Yaskawa INFORM job: SKRZYNIA_4740_0_STOPNI_2OBR.JBI

/JOB
//NAME SKRZYNIA_4740_0_STOPNI_2OBR
///FOLDERNAME 02-SKRZYNIE_JOBS
//POS
///NPOS 698,698,0,50,0,0
///TOOL 0
///POSTYPE PULSE
///PULSE
C00000=1055,-24125,84372,288,19725,204
C00001=0,-15438,65714,0,-68532,0
C00002=4718,-16587,59952,3396,-65485,-935
C00003=32997,-21499,42555,27623,-61436,21376
C00004=31759,-20688,42932,26837,-60850,21559
C00005=28987,-21156,42712,24818,-60442,22222
C00006=33447,-21964,42352,27886,-61721,21330
C00007=37687,-23357,41794,30651,-63289,20620
C00008=38979,-19018,48057,32961,-64962,20678
C00009=37261,-18075,48526,31902,-64209,20901
C00010=35830,-17198,48994,31015,-63571,21092
C00011=34080,-17614,48768,29780,-63290,21485
C00012=37261,-18075,48526,31902,-64209,20901
C00013=4718,-16587,59952,3396,-65485,-935
C00014=32997,-21499,42555,27623,-61436,21376
C00015=31759,-20688,42932,26837,-60850,21559
C00016=28987,-21156,42712,24818,-60442,22222
C00017=33447,-21964,42352,27886,-61721,21330
C00018=37687,-23357,41794,30651,-63289,20620
C00019=38979,-19018,48057,32961,-64962,20678
C00020=37261,-18075,48526,31902,-64209,20901
C00021=35830,-17198,48994,31015,-63571,21092
C00022=34080,-17614,48768,29780,-63290,21485
C00023=37261,-18075,48526,31902,-64209,20901
C00024=47373,-21912,40596,41149,-66086,26950
C00025=45033,-20851,41104,39798,-65001,27223
C00026=42790,-19693,41704,38494,-63946,27495
C00027=41070,-20182,41442,37324,-63566,27891
C00028=45033,-20851,41104,39798,-65001,27223
C00029=45033,-20851,41104,39798,-65001,27223
C00030=59624,-29540,14278,64846,-60867,16042
C00031=57357,-28542,14780,63940,-59509,16120
C00032=56188,-29140,14476,63237,-58995,16387
C00033=59588,-29370,14363,64862,-60819,16012
C00034=70875,-38414,-12574,117781,-105744,5605
C00035=70875,-38414,-12574,117781,-105744,5605
C00036=58486,-39981,-10562,86359,-50427,5279
C00037=56769,-35832,-2792,84059,-49443,6631
C00038=55152,-35009,-2405,83835,-48426,6454
C00039=53661,-35722,-2740,83085,-47530,6682
C00040=56769,-35832,-2792,84059,-49443,6631
C00041=87562,-48087,-13810,78020,-75252,11220
C00042=10104,-46603,4759,11228,-37390,-5046
C00043=0,-52280,40443,0,6876,0
C00044=1529,-42140,58025,-5964,2417,3265
C00045=0,-38374,23626,-1605,-51738,268
C00046=45044,-23015,37260,35797,-71879,25522
C00047=39973,-29571,18873,35060,-63052,24165
C00048=38620,-28701,19269,34339,-62304,24363
C00049=36409,-29254,19014,32896,-61805,24958
C00050=44451,-29039,21934,37281,-65892,23702
C00051=49472,-39353,6917,53118,-50908,20251
C00052=45058,-39356,3832,51653,-47640,20099
C00053=42883,-38319,4163,50577,-46309,20295
C00054=40255,-38926,3967,48502,-45334,21060
C00055=46774,-39679,3737,52663,-48537,19827
C00056=48708,-40455,3517,53615,-49689,19657
C00057=43798,-39237,3871,50850,-47027,20335
C00058=41951,-38324,4161,49930,-45891,20507
C00059=39836,-38844,3994,48234,-45126,21137
C00060=48489,-40338,3551,53521,-49551,19665
///LIMIT ON
C00061=1148,-56354,34370,-23,3827,-9
C00062=1148,-56354,34370,-23,3827,-9
///LIMIT OFF
C00063=48489,-40338,3551,53521,-49551,19665
C00064=44432,-39026,3936,51363,-47247,20139
C00065=42487,-38069,4248,50403,-46050,20315
C00066=39061,-38795,4009,47695,-44769,21310
C00067=44432,-39026,3936,51363,-47247,20139
C00068=43521,-36748,12770,50182,-45701,23408
C00069=41846,-35383,13175,49516,-44517,23399
C00070=39971,-34448,13485,48491,-43408,23582
C00071=37453,-34980,13306,46330,-42542,24334
C00072=41846,-35383,13175,49516,-44517,23399
C00073=78369,-41260,16071,67181,-65880,21417
C00074=137,-45861,52341,97,-67596,-14
C00075=-31499,-58302,-23356,15027,12889,-13082
C00076=-52768,-43016,-26078,18373,38595,-18774
C00077=-89470,-32103,-32973,29905,69139,-31512
C00078=-68838,-26884,-24872,16972,64732,-23076
C00079=-53036,-11528,-12218,12363,64665,-17409
C00080=-51536,-9474,-10276,11905,64649,-16876
C00081=-51739,-9114,-7787,12104,63269,-17104
C00082=-53036,-11528,-12218,12363,64665,-17409
C00083=-17541,-26226,-24397,927,59032,-5038
C00084=-17541,-26226,-24397,927,59032,-5038
C00085=-16950,-23991,-22741,715,59568,-4818
C00086=-17036,-23563,-20101,755,58071,-4857
C00087=-17541,-26226,-24397,927,59032,-5038
C00088=34102,-23192,-21614,-15638,64271,13209
C00089=33423,-21885,-20599,-15423,64418,12942
C00090=32426,-19856,-18975,-15106,64629,12551
C00091=32578,-19611,-17013,-15290,63535,12762
C00092=33423,-21885,-20599,-15423,64418,12942
C00093=59339,-6070,-6417,-20979,72191,20891
C00094=59339,-6070,-6417,-20979,72191,20891
C00095=57897,-4256,-4562,-20702,71913,20431
C00096=58108,-3992,-2506,-20878,70835,20713
C00097=59339,-6070,-6417,-20979,72191,20891
C00098=42744,-35904,-30225,-18322,62562,16651
C00099=-53036,-11528,-12218,12363,64665,-17409
C00100=-77982,-26538,-29134,27151,66629,-27745
C00101=-70983,-8594,-1966,26503,59809,-49670
C00102=-80152,19776,40785,37351,72704,-50428
C00103=-79984,20154,42529,37516,71911,-50638
C00104=-79233,18397,40079,37458,71885,-50340
C00105=-79984,20154,42529,37516,71911,-50638
C00106=-73519,23289,38838,28890,77081,-45618
C00107=-73519,24511,42682,29072,75582,-46027
C00108=-73519,23289,38838,28890,77081,-45618
C00109=-88897,15706,42282,50101,71325,-56974
C00110=-88897,15706,42282,50101,71325,-56974
C00111=-87612,12343,37838,50071,70996,-56519
C00112=-85283,14202,40272,50301,69633,-56165
C00113=-87338,12550,38107,50098,70839,-56476
C00114=-84952,-1789,13569,34660,47724,-58955
C00115=-67641,-1674,11109,10330,44856,-44725
C00116=-66443,961,13975,9688,44721,-44210
C00117=-67641,-1674,11109,10330,44856,-44725
C00118=-67641,-376,15347,10694,42950,-44967
C00119=-67641,-1674,11109,10330,44856,-44725
C00120=-79040,417,20398,15965,28992,-57786
C00121=-76655,5212,30978,15501,25024,-57306
C00122=-76655,6949,35816,16758,23084,-57955
C00123=-76655,5212,30978,15501,25024,-57306
C00124=-74761,6919,33010,13466,24593,-56049
C00125=-80460,-2874,12270,15804,32253,-57809
C00126=-61258,-29124,-13156,26560,43617,-22150
C00127=-30420,-40507,-29240,27153,53235,15188
C00128=-18589,-38725,-21450,23338,47896,18931
C00129=-17722,-35233,-16455,23322,46926,19051
C00130=-17722,-33749,-12435,23948,45421,18620
C00131=-17722,-33892,-12819,23887,45564,18661
C00132=-16677,-31133,-11209,23138,46167,19311
C00133=-17819,-35820,-17540,23246,47228,19090
C00134=-74104,-11494,-6266,31916,75042,4269
C00135=-71226,-7329,2631,32115,71468,4273
C00136=-71226,-6504,5446,32343,70365,3922
C00137=-71226,-6611,5086,32313,70505,3967
C00138=-68386,-4058,7675,32040,69573,4789
C00139=-73314,-9412,-353,32206,72648,3829
C00140=51751,-31069,-22965,-10739,49070,48663
C00141=49028,-23852,-11575,-9841,46366,47823
C00142=49028,-23004,-8935,-10039,45204,47956
C00143=49028,-23118,-9286,-10013,45357,47939
C00144=47000,-20813,-7527,-8928,45644,47024
C00145=50476,-26208,-15307,-10408,47325,48332
C00146=90602,-5375,6902,-38786,69848,59444
C00147=83174,19950,50269,-44999,67580,58220
C00148=82362,17902,47383,-44926,67511,57879
C00149=83515,19072,48341,-44798,68200,58056
C00150=78091,19382,40247,-36371,72286,52960
C00151=78091,20664,44011,-36670,70997,53443
C00152=78091,19382,40247,-36371,72286,52960
C00153=88699,7296,38566,-55615,63182,60372
C00154=86803,3068,32674,-55410,62638,59657
C00155=84852,4315,34115,-55564,61561,59330
C00156=86803,3068,32674,-55410,62638,59657
C00157=92770,-2803,21719,-53893,67577,59421
C00158=73393,-10627,10934,-27897,30744,62458
C00159=70789,-6606,18800,-27824,27830,62140
C00160=69654,-4593,20814,-26755,27596,61444
C00161=70789,-6606,18800,-27824,27830,62140
C00162=70789,-5070,23059,-29482,26284,63017
C00163=70789,-6606,18800,-27824,27830,62140
C00164=83486,-8736,6503,-27040,35338,66550
C00165=77831,-2041,26192,-25270,18452,68895
C00166=77967,1961,32070,-26860,17569,69698
C00167=77967,5243,40752,-32914,14549,72656
C00168=77967,1961,32070,-26860,17569,69698
C00169=74560,4730,35257,-21622,16551,66717
C00170=77967,1961,32070,-26860,17569,69698
C00171=81109,-22356,2664,-22493,33121,60116
C00172=86168,-49730,-13668,-23926,46819,49343
C00173=44183,-52048,-7537,-24795,46064,51426
C00174=0,-52280,40443,0,6876,0
C00175=0,-52280,40443,0,6876,0
C00176=33629,-57276,-6399,46271,-24969,-2804
C00177=75493,-63502,-64712,103874,-64610,-6298
C00178=48303,-58663,-62781,109560,-46378,-10551
C00179=44029,-59891,-64997,113806,-43206,-9136
C00180=55379,-67378,-68041,108237,-48773,-4935
C00181=62671,-64213,-64640,104431,-56093,-7372
C00182=28458,-50318,6850,47420,-25887,-3347
C00183=0,-52280,40443,0,6876,0
C00184=1055,-24125,84372,288,19725,204
C00185=0,-15438,65714,0,-68532,0
C00186=0,-15438,65714,966,-70097,42926
C00187=69988,-9219,57065,61610,-82752,27767
C00188=63113,-6157,59685,58080,-79692,28271
C00189=46529,-7301,64143,40614,-74233,29269
C00190=49501,-5951,66049,43527,-75687,29381
C00191=53417,-8187,64183,45775,-77170,28968
C00192=63113,-6157,59685,58080,-79692,28271
C00193=69988,-9219,57065,61610,-82752,27767
C00194=0,-15438,65714,966,-70097,42926
C00195=0,-15438,65714,0,-68532,0
C00196=1055,-24125,84372,288,19725,204
C00197=1055,-24125,84372,288,19725,204
C00198=0,-41971,13909,0,6774,1
C00199=-55064,-17017,13106,20113,45767,-35735
C00200=-85641,-3161,12660,31281,67420,-55579
C00201=-77611,9747,38455,32702,57795,-55547
C00202=-77611,9747,38455,32702,57795,-55547
C00203=-80481,23547,61641,37204,60115,-56891
C00204=-80479,11681,28780,33754,71138,-52780
C00205=-73572,15026,34389,33675,67405,-51294
C00206=-73572,20195,49236,35290,62248,-53161
C00207=-82806,26311,53816,38180,73291,-53604
C00208=-71695,3747,16001,30713,64750,-51022
C00209=-70421,5575,20105,30867,63066,-51036
C00210=-35543,-20105,-5144,22821,50284,-40173
C00211=-37830,-23193,-8618,23571,50957,-40982
C00212=11136,-28839,-12562,1025,41780,-20887
C00213=20486,-27077,-7346,-12554,38415,-10736
C00214=59545,-9921,5571,-27063,51925,3267
C00215=55110,-17412,-5825,-19778,50988,-2825
C00216=79390,11759,28162,-35512,71262,52960
C00217=74811,13878,33986,-35807,67493,52464
C00218=74942,18762,48004,-37392,62815,54352
C00219=76815,18630,46530,-37158,64288,54543
C00220=79390,11759,28162,-35512,71262,52960
C00221=10831,-54278,-29128,-6468,39852,-5090
C00222=-67200,-10549,24402,-3189,24913,-39001
C00223=-75122,-2194,12822,3152,39225,-43427
C00224=-77516,10189,32861,8493,33365,-45533
C00225=-75154,17575,49272,7885,27457,-44928
C00226=-68113,9932,38901,1157,28472,-40453
C00227=-67114,5383,31515,9208,32648,-43213
C00228=-66450,3998,29285,10896,33890,-43630
C00229=-66374,3101,28136,14657,35566,-44954
C00230=-66576,452,24763,27028,43375,-49112
C00231=-69928,4230,30673,35488,50431,-52676
C00232=-77050,-3138,8526,33226,61087,-51698
C00233=-67200,-10549,24402,-3189,24913,-39001
C00234=0,-52280,40443,83103,28146,-16510
C00235=99993,-20782,22705,-13349,24734,56519
C00236=67200,-10549,24402,3189,24913,39001
C00237=75122,-2194,12822,-3152,39225,43427
C00238=74323,5203,27259,-5972,33194,43789
C00239=74015,16414,48063,-6821,27325,44224
C00240=56519,1138,28747,9235,29393,33453
C00241=55467,619,28251,10155,29461,32830
C00242=56374,-724,25854,4078,30541,35419
C00243=56480,-7201,15910,-17697,38451,43334
C00244=68252,956,25699,-34035,49810,51639
C00245=77050,-3138,8526,-33226,61087,51698
C00246=67200,-10549,24402,3189,24913,39001
C00247=0,-52280,40443,-83103,28146,16510
C00248=-99993,-20782,22705,13349,24734,-56519
C00249=-91125,453,39555,30378,52425,-51131
C00250=-81425,-5449,14825,37552,56592,-47667
C00251=-81425,-10835,-2515,34915,62871,-45127
C00252=-79239,4305,16082,37593,68846,-50182
C00253=-81302,5892,27588,46359,62943,-54679
C00254=-82227,19402,59913,51524,57300,-60581
C00255=-84844,8890,27031,38640,69740,-53449
C00256=-90096,4679,14083,37467,76581,-51973
C00257=-87885,29238,52923,40761,81198,69685
C00258=-84355,23847,39024,40698,83720,72224
C00259=-81960,27335,46957,41070,80536,71891
C00260=-82643,24718,50492,48951,72637,70260
C00261=-90480,18737,31939,47254,81986,71631
C00262=-94217,10634,17426,46901,86469,-59967
C00263=-81425,-10835,-2515,34915,62871,-45127
C00264=-81425,-5449,14825,37552,56592,-47667
C00265=-94290,-610,44819,32366,49686,-53459
C00266=0,-55136,17047,60468,32096,-4233
C00267=99993,-20782,22705,-13349,24734,56519
C00268=91125,453,39555,-30378,52425,51131
C00269=81425,-5449,14825,-37552,56592,47667
C00270=81425,-10835,-2515,-34915,62871,45127
C00271=79239,4305,16082,-37593,68846,50182
C00272=83239,4964,30263,-50637,62037,57149
C00273=83991,16425,61235,-57769,55250,63273
C00274=93928,7973,40920,-53095,64494,61640
C00275=75109,22299,39152,-26915,78743,47998
C00276=79256,17348,34699,-33448,76412,88212
C00277=79932,23608,50901,-39863,71219,88955
C00278=76220,30771,63034,-41386,67395,88927
C00279=86322,16060,37848,-39554,76452,89287
C00280=87424,-1569,9538,-38190,72401,52253
C00281=81425,-10835,-2515,-34915,62871,45127
C00282=92850,-11266,9233,-39092,60986,50964
C00283=28366,-40369,19479,-5635,23506,17663
C00284=-80334,-19501,31260,21216,42469,-40219
C00285=-80621,-32280,-9061,25825,59412,-41877
C00286=-80621,-37319,-22868,24573,64555,-40576
C00287=-75108,-2453,16462,35304,60348,-42510
C00288=-72231,7240,33473,36511,55681,-43130
C00289=-35770,-19109,7486,28512,40799,-31761
C00290=-39606,-22901,-1163,28356,44724,-32188
C00291=15344,-29112,-5358,-2858,33820,-6852
C00292=13390,-24012,2637,-1527,32105,-7853
C00293=57983,-8601,15571,-27088,42703,12849
C00294=60973,-17187,4937,-27817,44388,13718
C00295=60973,-17187,4937,-27817,44388,13718
C00296=-13287,-42463,-12044,19170,31021,-23010
C00297=-17374,-21287,20534,22794,29118,-26096
C00298=13276,-20759,18622,-1911,29377,-7028
C00299=39924,-14247,19329,-14795,35999,4396
C00300=41528,-14133,18797,-15449,36702,5040
C00301=57001,-5890,26499,-21893,40771,11494
C00302=64054,-19541,3059,-29141,44956,15011
C00303=51466,-33957,-1499,-46586,51805,23434
C00304=17032,-20770,22044,-28854,30468,11088
C00305=-9868,-18638,14971,-8492,38486,-5199
C00306=-40562,-13194,19800,9508,35447,-20184
C00307=-41848,-12620,20103,10165,35810,-20773
C00308=-57278,-4046,28217,17578,39066,-27653
C00309=-71680,-19835,10874,33863,39440,-36917
C00310=-20806,-37586,-12792,9951,42782,-18031
C00311=29087,-45372,27330,-13325,19529,9021
C00312=0,-52280,40443,0,6876,0
C00313=0,-52280,40443,0,6876,0
C00314=0,-52280,40443,0,6876,0
C00315=0,-52280,40443,0,-40718,0
C00316=32359,-35955,27464,28918,-49457,29587
C00317=33244,-30989,28192,31082,-46894,28340
C00318=17779,-48456,-23364,103225,-11582,-7642
C00319=21302,-27483,32723,20378,-44693,31826
C00320=26032,-39616,1147,25257,-48263,28480
C00321=26032,-42284,-4858,26096,-46359,27892
C00322=29904,-46498,-2819,27004,-47536,28031
C00323=45803,-31685,22885,64496,-39050,18987
C00324=0,-52277,40442,0,6872,2
///LIMIT ON
C00325=0,-38538,66749,0,-898,0
///LIMIT OFF
C00326=0,-52280,40443,0,-79033,35417
C00327=63837,-43435,-10267,65210,-58810,8342
C00328=51738,-38814,-970,57660,-53573,11589
C00329=47613,-40374,-5302,59887,-48365,10192
C00330=46201,-27302,20507,44767,-62342,18270
C00331=53914,-29436,22058,48262,-67266,17843
C00332=63113,-6157,59685,58080,-79692,28271
C00333=53636,-7999,65947,44587,-77595,28821
C00334=47087,-5642,67901,40734,-75391,29611
C00335=49534,-5270,67671,43393,-76105,29552
C00336=58547,-7653,65645,48613,-79176,28479
C00337=0,-52280,40443,0,-79033,35417
C00338=0,-38922,70509,0,-71891,28081
C00339=0,-38922,70509,0,-71891,28081
C00340=36958,-10079,72709,30464,-66560,20948
C00341=30207,-8205,71936,26080,-63666,21556
C00342=5819,-37145,831,436,-53029,28466
C00343=13946,-45192,10090,9828,-39459,25958
///LIMIT ON
C00344=404,-42897,57020,-1574,2523,869
///LIMIT OFF
C00345=0,-52280,40443,0,6876,0
C00346=-99253,-13690,44082,59847,13407,-31313
C00347=-87814,-12734,20141,45739,-14352,-64418
C00348=-86669,-6582,30812,41148,-16781,-62025
C00349=-85055,-5827,31548,44003,-17420,-63187
C00350=-85971,-6262,31124,42409,-17052,-62539
C00351=-86650,-5303,32069,41395,-16716,-62141
C00352=-94954,-14494,-1860,-7818,15857,-59130
C00353=-94509,1544,30797,-849,15127,-60471
C00354=-94509,4151,37772,-1041,12286,-60378
C00355=-88011,-10036,27574,37950,-16527,-60658
C00356=-86125,-12470,22545,29004,-25567,-58412
C00357=-85732,-21202,11427,30682,-24763,-59235
C00358=-84150,-10929,23786,31981,-25941,-59678
C00359=-83036,-10419,24246,33504,-26268,-60308
C00360=-84150,-10929,23786,31981,-25941,-59678
C00361=-85291,-9507,25078,30650,-25411,-59154
C00362=-84150,-10929,23786,31981,-25941,-59678
C00363=-85786,-16909,14677,31743,-23900,-59790
C00364=-84150,-10498,24888,31517,-26306,-59436
C00365=-83174,-10052,25293,32841,-26587,-59984
C00366=-84150,-10498,24888,31517,-26306,-59436
C00367=-85258,-9112,26156,30226,-25800,-58928
C00368=-84150,-10498,24888,31517,-26306,-59436
C00369=-87841,-18519,13420,28367,-23534,-58339
C00370=-84150,-10465,24972,31484,-26336,-59417
C00371=-83241,-10052,25348,32714,-26598,-59924
C00372=-84150,-10465,24972,31484,-26336,-59417
C00373=-85145,-9228,26102,30329,-25881,-58963
C00374=-84150,-10465,24972,31484,-26336,-59417
C00375=-86371,-18277,13606,30568,-23951,-59265
C00376=-84345,-11688,21985,32461,-25312,-59957
C00377=-83211,-11173,22442,34044,-25650,-60618
C00378=-84345,-11688,21985,32461,-25312,-59957
C00379=-85283,-10526,23025,31366,-24861,-59525
C00380=-84345,-11688,21985,32461,-25312,-59957
C00381=-86191,-19647,12567,30467,-24278,-59187
C00382=-84345,-10877,24073,31552,-26006,-59481
C00383=-83051,-10286,24607,33321,-26381,-60213
C00384=-84345,-10877,24073,31552,-26006,-59481
C00385=-85179,-9842,25009,30582,-25619,-59100
C00386=-84345,-10877,24073,31552,-26006,-59481
C00387=-85438,-18022,14839,31140,-24818,-59429
C00388=-84247,-11820,22550,32049,-25753,-59727
C00389=-84104,-10976,23642,32111,-25899,-59738
C00390=-82990,-10465,24105,33639,-26227,-60372
C00391=-84104,-10976,23642,32111,-25899,-59738
C00392=-84898,-9998,24525,31196,-25529,-59378
C00393=-84104,-10976,23642,32111,-25899,-59738
C00394=-86610,-16845,14732,30573,-23614,-59301
C00395=-84104,-10864,23927,31990,-25993,-59674
C00396=-82824,-10273,24459,33737,-26370,-60397
C00397=-84104,-10864,23927,31990,-25993,-59674
C00398=-84789,-10021,24690,31200,-25673,-59363
C00399=-84104,-10864,23927,31990,-25993,-59674
C00400=-83806,-19585,12613,33764,-25080,-60559
C00401=-83924,-10205,25475,31619,-26533,-59453
C00402=-82780,-9675,25960,33156,-26866,-60087
C00403=-83924,-10205,25475,31619,-26533,-59453
C00404=-84478,-9530,26093,30986,-26280,-59206
C00405=-83924,-10205,25475,31619,-26533,-59453
C00406=-87149,-17993,13826,29513,-23647,-58830
C00407=-84920,-13182,20975,31162,-25481,-59361
C00408=-83711,-10572,24852,32056,-26475,-59649
C00409=-82779,-10142,25241,33309,-26748,-60166
C00410=-83711,-10572,24852,32056,-26475,-59649
C00411=-84370,-9774,25579,31305,-26170,-59356
C00412=-83711,-10572,24852,32056,-26475,-59649
C00413=-83642,-3679,42021,23358,-36761,-56118
C00414=-85886,-5975,41264,18964,-40261,-54782
C00415=-83919,-11632,22322,32811,-25616,-60079
C00416=-82884,-11162,22742,34234,-25925,-60671
C00417=-83919,-11632,22322,32811,-25616,-60079
C00418=-84723,-10654,23196,31887,-25230,-59715
C00419=-83919,-11632,22322,32811,-25616,-60079
C00420=-87348,-16035,7353,17528,-35245,-56477
C00421=-86244,-15062,8172,18754,-35315,-57058
C00422=-86244,-16649,3638,19674,-33501,-57585
C00423=-85308,-16228,3988,20718,-33648,-58082
C00424=-86244,-16649,3638,19674,-33501,-57585
C00425=-86740,-15973,4201,19194,-33277,-57362
C00426=-86244,-16649,3638,19674,-33501,-57585
C00427=-73780,-8639,20128,34258,-51705,-52097
C00428=-90711,-17528,-28778,11328,-28245,-57111
C00429=-92565,-19610,-33223,7138,-24591,-57051
C00430=-91512,-19116,-32812,8551,-24603,-57834
C00431=-92565,-19610,-33223,7138,-24591,-57051
C00432=-93003,-18716,-32476,6600,-24397,-56752
C00433=-92565,-19610,-33223,7138,-24591,-57051
C00434=-92565,-19610,-33223,7138,-24591,-57051
C00435=-95836,-54375,-51122,6031,-17685,-48210
C00436=-95836,-54375,-51122,6031,-17685,-48210
C00437=-71303,-59965,-23787,8701,20788,-26710
C00438=-43821,-47238,-2775,-3022,56549,-3681
C00439=-20126,-26882,59542,2406,16879,-9162
C00440=-20126,-26882,59542,2406,16879,-9162
C00441=98601,-10520,92678,4674,-40855,-9615
C00442=95537,-19831,-2695,-2933,-44471,35837
C00443=92548,-20391,-28429,-6186,-30623,55200
C00444=91429,-17018,-28974,-8057,-27827,56250
C00445=91429,-17018,-28974,-8057,-27827,56250
C00446=90371,-16495,-28521,-9286,-27856,56953
C00447=91429,-17018,-28974,-8057,-27827,56250
C00448=92033,-15799,-27911,-7415,-27588,55880
C00449=91429,-17018,-28974,-8057,-27827,56250
C00450=92548,-20391,-28429,-6186,-30623,55200
C00451=91156,-15018,-4648,-8036,-38181,54813
C00452=90585,-14766,-4428,-8565,-38201,55100
C00453=88830,-13959,-3717,-10186,-38284,55977
C00454=89897,-14456,-4157,-9202,-38230,55445
C00455=90761,-12944,-2809,-8452,-37927,55043
C00456=89897,-14456,-4157,-9202,-38230,55445
C00457=89670,-8466,73559,-9449,-60959,55261
C00458=89910,-11217,67535,-9455,-58896,55399
C00459=85786,-16735,14816,-31782,-23869,59812
C00460=83514,-12996,17929,-35760,-24132,61552
C00461=82251,-12406,18443,-37550,-24551,62308
C00462=83514,-12996,17929,-35760,-24132,61552
C00463=84258,-12095,18717,-34917,-23742,61217
C00464=83514,-12996,17929,-35760,-24132,61552
C00465=87149,-17993,13826,-29513,-23647,58830
C00466=83118,-12818,18089,-36330,-24263,61791
C00467=81915,-12248,18589,-38020,-24666,62504
C00468=83118,-12818,18089,-36330,-24263,61791
C00469=83897,-11882,18912,-35460,-23856,61445
C00470=83118,-12818,18089,-36330,-24263,61791
C00471=83806,-19585,12613,-33764,-25080,60559
C00472=82998,-13006,17925,-36445,-24332,61826
C00473=81675,-12378,18472,-38297,-24777,62607
C00474=82998,-13006,17925,-36445,-24332,61826
C00475=83876,-11958,18841,-35466,-23874,61442
C00476=82998,-13006,17925,-36445,-24332,61826
C00477=86610,-16845,14732,-30573,-23614,59301
C00478=82493,-13239,17725,-37070,-24559,62089
C00479=81406,-12724,18174,-38578,-24928,62723
C00480=82493,-13239,17725,-37070,-24559,62089
C00481=83436,-12134,18690,-36041,-24064,61684
C00482=82493,-13239,17725,-37070,-24559,62089
C00483=84814,-16043,15376,-33312,-24093,60464
C00484=82555,-13613,17404,-36910,-24580,62015
C00485=81384,-13062,17878,-38534,-24974,62698
C00486=82555,-13613,17404,-36910,-24580,62015
C00487=83566,-12434,18427,-35805,-24047,61580
C00488=82555,-13613,17404,-36910,-24580,62015
C00489=86191,-19647,12567,-30467,-24278,59187
C00490=82500,-13648,17375,-36975,-24607,62039
C00491=81467,-13161,17792,-38413,-24955,62645
C00492=82500,-13648,17375,-36975,-24607,62039
C00493=83481,-12505,18364,-35905,-24087,61617
C00494=82500,-13648,17375,-36975,-24607,62039
C00495=86371,-18277,13606,-30568,-23951,59265
C00496=82904,-13790,17251,-36416,-24470,61808
C00497=81715,-13237,17726,-38081,-24865,62509
C00498=82904,-13790,17251,-36416,-24470,61808
C00499=83686,-12878,18037,-35556,-24055,61469
C00500=82904,-13790,17251,-36416,-24470,61808
C00501=87841,-18519,13420,-28367,-23534,58339
C00502=82748,-13879,17174,-36603,-24542,61883
C00503=81692,-13388,17594,-38077,-24893,62505
C00504=82748,-13879,17174,-36603,-24542,61883
C00505=83607,-12881,18032,-35663,-24082,61515
C00506=82748,-13879,17174,-36603,-24542,61883
C00507=85786,-16909,14677,-31743,-23900,59790
C00508=82520,-14198,16902,-36833,-24674,61972
C00509=81460,-13708,17319,-38301,-25026,62591
C00510=82520,-14198,16902,-36833,-24674,61972
C00511=83571,-12989,17938,-35691,-24113,61524
C00512=82520,-14198,16902,-36833,-24674,61972
C00513=85732,-21202,11427,-30682,-24763,59235
C00514=82398,-14365,16763,-36952,-24745,62014
C00515=81172,-13798,17245,-38643,-25153,62725
C00516=82398,-14365,16763,-36952,-24745,62014
C00517=83600,-12984,17944,-35650,-24102,61504
C00518=82398,-14365,16763,-36952,-24745,62014
C00519=86140,-12802,12665,-93523,-10743,85795
C00520=86140,-12802,12665,-93523,-10743,85795
C00521=85030,-12289,13120,-93723,-11463,85776
C00522=86140,-12802,12665,-93523,-10743,85795
C00523=86958,-11660,13681,-94506,-10238,86349
C00524=85239,-16743,-4327,42764,21357,45785
C00525=86674,107,23869,25042,24033,51593
C00526=86674,2327,30134,27824,21680,50173
C00527=87715,-15254,10554,-91589,-9692,85040
C00528=85045,-36869,-4353,-28502,-22832,52282
C00529=0,-24029,84339,0,19981,0
C00530=0,-24029,84339,0,19981,0
C00531=3172,-24246,80980,3465,15913,689
C00532=-86563,-26985,13879,10257,-21548,-45530
C00533=-86191,-19647,12567,30467,-24278,-59187
C00534=-83221,-13587,17636,37793,-25116,-62228
C00535=-91978,-13833,14560,12391,-18633,-51524
C00536=-94992,-13830,14285,1276,-18012,-46664
C00537=-84074,-17488,11256,38660,-23649,-62784
C00538=-73679,-33270,1000,44272,-31600,-64253
///LIMIT ON
C00539=-86926,-60758,23267,6576,1160,-9545
///LIMIT OFF
C00540=0,-52280,40443,0,6876,0
///LIMIT ON
C00541=82475,-58079,26734,835,4084,4444
///LIMIT OFF
C00542=97932,-26840,7691,8784,-23444,42538
C00543=87166,-16607,16322,-25365,-24201,56345
C00544=84699,-11354,21752,-29145,-24735,57949
C00545=84804,-11023,22730,-28561,-25071,57659
C00546=85100,-26994,10417,-24982,-28140,55821
C00547=0,-52280,40443,0,6876,0
C00548=0,-52280,40443,0,6876,0
///LIMIT ON
C00549=-90140,-60305,18108,-2708,1721,-7625
///LIMIT OFF
C00550=-95594,-27428,6866,-4663,-19832,-42154
C00551=-98688,-13767,16447,-18366,-10080,-35766
C00552=-98967,-3050,34440,-28957,-8622,-29685
C00553=-100063,5316,51567,-32262,-10006,-27560
C00554=-94586,18541,64268,-6451,10518,-43578
C00555=-95535,2380,25473,239,27557,-47214
C00556=-91259,3120,34463,-5130,22041,-43946
C00557=-95333,12702,45733,36,21375,-47085
C00558=-99268,-13088,27343,-18620,-14105,-35021
///LIMIT ON
C00559=-90140,-60305,18108,-2708,1721,-7625
///LIMIT OFF
C00560=0,-52280,40443,0,6876,0
///LIMIT ON
C00561=84259,-57935,27522,-3761,3673,6310
///LIMIT OFF
C00562=86507,-39672,4297,-27618,-16640,46340
C00563=73669,-37119,-20783,-92053,-19719,85232
C00564=86539,-20830,1725,-71850,-11773,76853
C00565=90325,-18913,6238,-62161,-7452,70888
///LIMIT ON
C00566=97679,-11879,12650,-55334,4229,66281
///LIMIT OFF
C00567=98389,-8856,11720,-15676,14634,48538
C00568=96255,-748,20886,-3277,24061,38276
C00569=95132,-6008,10010,1655,28777,36730
C00570=94050,-4188,7205,-2481,41508,36662
C00571=98126,4908,16834,-5042,41918,38535
C00572=100487,-9453,-1206,-10413,41328,41147
C00573=96250,-19428,-8283,-4838,27297,37910
C00574=86507,-39672,4297,-27618,-16640,46340
///LIMIT ON
C00575=84259,-57935,27522,-3761,3673,6310
///LIMIT OFF
C00576=0,-52280,40443,0,6876,0
C00577=0,-27933,77061,0,20812,0
C00578=0,-27933,77061,0,20812,0
C00579=0,-52280,40443,0,6876,0
///LIMIT ON
C00580=-91970,-60791,14435,-3343,512,-9412
///LIMIT OFF
C00581=-98647,-24138,10005,-11519,-21203,-39749
C00582=-99883,-13980,22886,-11640,-25090,-40341
C00583=-99702,-9154,61728,-1148,-61809,-40243
C00584=-84328,-13042,29707,23458,-33731,-54641
C00585=-83101,-4179,39208,25894,-34785,-55667
C00586=-82881,-4330,38692,26392,-34479,-55866
C00587=-76259,-18287,26646,31659,-38322,-57579
C00588=-89741,-28009,12101,4461,-28076,-46404
///LIMIT ON
C00589=-91970,-60791,14435,-3343,512,-9412
///LIMIT OFF
C00590=0,-52280,40443,0,6876,0
///LIMIT ON
C00591=91083,-60784,14823,-9043,-825,15173
///LIMIT OFF
C00592=83869,-19403,12921,-33769,-24740,60260
C00593=83869,-19403,12921,-33769,-24740,60260
C00594=83932,-19538,53415,-33663,-71112,60249
C00595=83932,-19538,53415,-33663,-71112,60249
C00596=82480,-12247,21118,-35440,-26416,60009
C00597=82194,-11433,19802,-37650,-25323,61125
C00598=81904,-9374,24711,-35791,-26879,60109
C00599=79790,-20261,14917,-36681,-28829,60258
C00600=76554,-29711,-1870,-46042,-25952,65654
///LIMIT ON
C00601=91083,-60784,14823,-9043,-825,15173
///LIMIT OFF
C00602=0,-52280,40443,0,6876,0
///LIMIT ON
C00603=-91526,-60598,16699,7584,176,-13289
///LIMIT OFF
C00604=-81382,-25890,9219,35455,-25500,-59095
C00605=-86453,-20958,12525,30076,-22568,-57089
C00606=-86589,-16097,16237,31250,-21582,-57704
C00607=-98933,-11298,20505,-13970,-18736,-37953
C00608=-98281,-10965,21163,-11559,-18548,-39330
C00609=-85424,-18472,14402,34409,-22969,-58895
C00610=-74746,-27148,8488,44263,-29128,-62418
C00611=-81326,-27507,8265,35533,-26282,-59001
///LIMIT ON
C00612=-91415,-60262,16631,7870,-73,-13734
///LIMIT OFF
C00613=24,-24029,84339,7,19981,5
C00614=100404,-52373,45687,-1822,14816,-5144
C00615=75939,-26469,7919,-40869,-29645,63133
C00616=81882,-22565,10470,-35355,-26404,61107
C00617=82801,-12246,21732,-34208,-26055,60642
C00618=91824,-10567,23615,-8659,-22197,49820
C00619=96485,-9539,26282,5686,-23135,43736
C00620=77262,-23244,14300,-38922,-31295,61912
C00621=96357,-33562,33410,58602,-23427,10353
C00622=568,-24029,84339,168,19981,112
///LIMIT ON
C00623=-91970,-60791,14435,-3343,512,-9412
///LIMIT OFF
C00624=-98991,-22833,11519,-12824,-17638,-36336
C00625=-86376,-13627,18436,38326,-18406,-58533
C00626=-85581,-10814,20279,41280,-18093,-59893
C00627=-85561,-10517,20811,41029,-18209,-59765
C00628=-86274,-24518,9978,34497,-20333,-56613
C00629=-91684,-53777,2301,20525,-9313,-33684
C00630=-67305,-55044,34987,1504,5690,-2468
C00631=0,-52280,40443,0,6876,0
///LIMIT ON
C00632=77036,-56616,31288,-2531,4707,4197
///LIMIT OFF
C00633=84359,-28321,8817,-32860,-20485,54199
C00634=81156,-16932,14874,-39538,-26422,62851
C00635=93321,-15690,11640,-5466,-17578,48664
C00636=91404,-14588,14576,-11730,-19131,51290
C00637=77970,-27630,4721,-41834,-28549,63607
C00638=81111,-35571,7141,-33980,-21909,52006
///LIMIT ON
C00639=82490,-55811,26416,-6832,1088,10458
///LIMIT OFF
C00640=0,-52280,40443,0,6876,0
C00641=0,-28135,76691,0,20839,0
C00642=0,-28135,76691,0,20839,0
C00643=-45332,-39712,59352,-1730,18713,2903
C00644=-94065,-8316,59352,-1730,-37754,-40387
C00645=-100331,-14895,33931,-8215,-36518,-40227
C00646=-98931,-8578,39429,-6260,-48307,-43744
C00647=-100336,-4176,46216,-7600,-55875,-44633
C00648=-93952,8947,73671,995,-68520,-43850
C00649=-98791,-3170,32594,-4861,-60761,-43748
C00650=-98723,4324,37855,-4919,-58743,-43677
C00651=-98691,-12730,-17828,-7584,-33364,-41886
C00652=-98599,-14408,-28132,-8909,-27584,-41168
C00653=-99605,-15546,-21493,-8548,-33053,-41326
C00654=-98632,914,40428,-4141,-58435,-42510
C00655=-93952,8947,73671,995,-68520,-43850
C00656=-88754,54,62805,4404,-67858,-45120
C00657=-100222,-4532,45667,-7492,-55263,-44561
C00658=-100331,-14895,33931,-8215,-36518,-40227
C00659=-94065,-8316,59352,-1730,-37754,-40387
C00660=-45544,-32973,71870,-2133,15168,3033
C00661=0,-28135,76691,0,20839,0
C00662=54178,-17846,77779,596,-29686,20997
C00663=54178,-17846,77779,596,-29686,20997
C00664=99462,-18987,75418,611,-28919,20989
C00665=98707,-9390,78674,1080,-71212,38250
C00666=98768,-5182,41096,1808,-44974,38308
C00667=100431,1771,51615,3823,-56746,39115
C00668=97953,-6621,17555,2289,-50176,39420
C00669=95834,-5353,18817,760,-50052,40242
C00670=86579,-3733,19265,-13263,-48799,44764
C00671=89140,-11519,-8899,-11291,-36869,46482
C00672=89026,-14065,-21014,-13447,-30614,47708
C00673=90457,-16080,-12990,-9972,-37305,45724
C00674=97953,-6621,17555,2289,-50176,39420
C00675=100431,1771,51615,3823,-56746,39115
C00676=98768,-5182,41096,1808,-44974,38308
C00677=98707,-9390,78674,1080,-71212,38250
C00678=0,-28135,76691,0,20839,0
C00679=0,-28135,76691,0,20839,0
///LIMIT ON
C00680=-91526,-60598,16699,7584,176,-13289
///LIMIT OFF
C00681=-81382,-25890,9219,35455,-25500,-59095
C00682=-81382,-25890,9219,35455,-25500,-59095
C00683=-85509,-13950,19358,32213,-22393,-58041
C00684=-96341,-12327,18855,-5124,-17594,-42111
C00685=-97523,-9822,24708,-8570,-19966,-40659
C00686=-84656,-25369,12054,31249,-26195,-57129
///LIMIT ON
C00687=-82652,-57346,29982,2770,3944,-5064
///LIMIT OFF
C00688=0,-52280,40443,0,6876,0
C00689=60653,-54633,35892,-1212,5841,2035
C00690=77942,-28227,6869,-38010,-29303,61907
C00691=82500,-13648,17375,-36975,-24607,62039
C00692=80731,-11587,18684,-41654,-25449,63953
C00693=80409,-10373,22284,-40214,-26848,63104
C00694=64389,-31987,5108,-50419,-37074,66126
C00695=60653,-54633,35892,-1212,5841,2035
C00696=0,-52280,40443,0,6876,0
C00697=0,-28167,76633,0,20843,0
BC00000=428499
BC00001=428499
BC00002=311358
BC00003=264574
BC00004=264574
BC00005=264574
BC00006=264574
BC00007=233852
BC00008=299649
BC00009=299649
BC00010=299649
BC00011=299649
BC00012=299649
BC00013=403524
BC00014=372101
BC00015=372101
BC00016=372101
BC00017=372101
BC00018=372101
BC00019=422537
BC00020=422537
BC00021=422537
BC00022=422537
BC00023=422537
BC00024=494794
BC00025=494794
BC00026=494794
BC00027=494794
BC00028=494794
BC00029=545598
BC00030=545598
BC00031=545598
BC00032=545598
BC00033=545598
BC00034=499632
BC00035=616274
BC00036=594322
BC00037=594322
BC00038=594322
BC00039=594322
BC00040=594322
BC00041=569159
BC00042=503930
BC00043=490792
BC00044=671734
BC00045=689202
BC00046=704563
BC00047=704563
BC00048=704563
BC00049=704563
BC00050=704563
BC00051=741824
BC00052=741824
BC00053=741824
BC00054=741824
BC00055=741824
BC00056=791630
BC00057=788281
BC00058=788281
BC00059=788281
BC00060=788281
BC00061=667682
BC00062=808508
BC00063=874870
BC00064=865782
BC00065=865782
BC00066=865782
BC00067=865782
BC00068=895576
BC00069=886359
BC00070=886359
BC00071=886359
BC00072=886359
BC00073=895757
BC00074=866045
BC00075=927819
BC00076=927819
BC00077=927819
BC00078=943180
BC00079=943180
BC00080=943180
BC00081=943180
BC00082=943180
BC00083=943180
BC00084=943180
BC00085=943180
BC00086=943180
BC00087=943180
BC00088=943180
BC00089=943180
BC00090=943180
BC00091=943180
BC00092=943180
BC00093=943180
BC00094=943180
BC00095=943180
BC00096=943180
BC00097=943180
BC00098=943180
BC00099=943180
BC00100=943180
BC00101=943180
BC00102=943180
BC00103=943182
BC00104=943182
BC00105=943182
BC00106=943182
BC00107=943182
BC00108=943182
BC00109=943182
BC00110=943182
BC00111=943182
BC00112=943182
BC00113=943182
BC00114=943182
BC00115=943182
BC00116=943182
BC00117=943182
BC00118=943182
BC00119=943182
BC00120=943182
BC00121=943182
BC00122=943182
BC00123=943182
BC00124=943182
BC00125=943182
BC00126=943183
BC00127=943184
BC00128=943184
BC00129=943184
BC00130=943184
BC00131=943184
BC00132=943184
BC00133=943184
BC00134=943184
BC00135=943184
BC00136=943184
BC00137=943184
BC00138=943156
BC00139=943170
BC00140=943170
BC00141=943170
BC00142=943170
BC00143=943170
BC00144=943170
BC00145=943170
BC00146=943184
BC00147=943184
BC00148=943184
BC00149=943184
BC00150=943184
BC00151=943184
BC00152=943184
BC00153=943184
BC00154=943184
BC00155=943184
BC00156=943184
BC00157=943184
BC00158=943184
BC00159=943184
BC00160=943184
BC00161=943184
BC00162=943184
BC00163=943184
BC00164=943184
BC00165=943184
BC00166=943184
BC00167=943184
BC00168=943184
BC00169=943184
BC00170=943184
BC00171=911399
BC00172=884954
BC00173=838173
BC00174=838173
BC00175=665258
BC00176=749913
BC00177=766195
BC00178=766198
BC00179=824721
BC00180=827288
BC00181=710557
BC00182=681076
BC00183=705154
BC00184=428499
BC00185=428499
BC00186=428499
BC00187=423987
BC00188=423987
BC00189=424111
BC00190=362753
BC00191=362753
BC00192=423987
BC00193=423987
BC00194=428499
BC00195=428499
BC00196=428499
BC00197=520863
BC00198=893917
BC00199=915147
BC00200=918406
BC00201=918406
BC00202=918406
BC00203=918406
BC00204=935268
BC00205=935270
BC00206=935270
BC00207=935270
BC00208=935270
BC00209=935270
BC00210=935270
BC00211=935270
BC00212=935270
BC00213=935269
BC00214=935270
BC00215=935271
BC00216=935271
BC00217=935271
BC00218=935271
BC00219=935271
BC00220=935271
BC00221=930781
BC00222=906929
BC00223=936106
BC00224=936109
BC00225=936109
BC00226=936106
BC00227=936107
BC00228=936108
BC00229=936108
BC00230=936109
BC00231=936109
BC00232=936109
BC00233=906929
BC00234=835535
BC00235=835535
BC00236=906929
BC00237=936106
BC00238=936109
BC00239=936109
BC00240=936109
BC00241=936109
BC00242=936114
BC00243=936121
BC00244=936110
BC00245=936109
BC00246=906929
BC00247=835535
BC00248=835535
BC00249=872997
BC00250=918800
BC00251=938197
BC00252=938199
BC00253=938199
BC00254=938199
BC00255=938199
BC00256=938775
BC00257=938199
BC00258=952138
BC00259=952138
BC00260=952138
BC00261=952138
BC00262=952138
BC00263=938197
BC00264=918800
BC00265=872997
BC00266=873283
BC00267=835535
BC00268=872997
BC00269=918800
BC00270=938197
BC00271=938199
BC00272=938199
BC00273=938199
BC00274=938199
BC00275=938199
BC00276=938199
BC00277=938199
BC00278=938199
BC00279=938199
BC00280=938199
BC00281=938197
BC00282=918800
BC00283=849812
BC00284=864290
BC00285=883850
BC00286=922155
BC00287=922155
BC00288=922155
BC00289=922153
BC00290=922155
BC00291=922155
BC00292=922155
BC00293=922153
BC00294=922155
BC00295=914820
BC00296=922155
BC00297=922155
BC00298=922151
BC00299=922153
BC00300=922197
BC00301=922153
BC00302=922155
BC00303=922155
BC00304=922151
BC00305=922153
BC00306=922155
BC00307=922155
BC00308=922155
BC00309=922155
BC00310=918747
BC00311=805523
BC00312=697681
BC00313=713042
BC00314=778618
BC00315=824674
BC00316=898714
BC00317=898714
BC00318=898714
BC00319=898714
BC00320=901485
BC00321=889045
BC00322=898714
BC00323=860475
BC00324=785682
BC00325=523177
BC00326=523177
BC00327=561362
BC00328=561362
BC00329=561362
BC00330=508601
BC00331=507340
BC00332=301099
BC00333=301226
BC00334=300802
BC00335=256793
BC00336=256782
BC00337=523177
BC00338=523177
BC00339=661219
BC00340=661219
BC00341=661219
BC00342=661219
BC00343=661219
BC00344=602144
BC00345=753376
BC00346=785096
BC00347=886828
BC00348=886828
BC00349=886828
BC00350=886828
BC00351=886828
BC00352=886828
BC00353=886828
BC00354=886828
BC00355=886828
BC00356=886828
BC00357=917549
BC00358=910733
BC00359=910733
BC00360=910733
BC00361=910733
BC00362=910733
BC00363=856105
BC00364=856105
BC00365=856105
BC00366=856105
BC00367=856105
BC00368=856105
BC00369=794661
BC00370=786693
BC00371=786693
BC00372=786693
BC00373=786693
BC00374=786693
BC00375=733216
BC00376=733216
BC00377=733216
BC00378=733216
BC00379=733216
BC00380=733216
BC00381=671766
BC00382=664534
BC00383=664534
BC00384=664534
BC00385=664534
BC00386=664534
BC00387=610322
BC00388=610322
BC00389=610322
BC00390=610322
BC00391=610322
BC00392=610322
BC00393=610322
BC00394=548878
BC00395=540590
BC00396=540590
BC00397=540590
BC00398=540590
BC00399=540590
BC00400=487434
BC00401=487434
BC00402=487434
BC00403=487434
BC00404=487434
BC00405=487434
BC00406=425990
BC00407=421023
BC00408=418329
BC00409=418329
BC00410=418329
BC00411=418329
BC00412=418329
BC00413=418329
BC00414=364547
BC00415=364547
BC00416=364547
BC00417=364547
BC00418=364547
BC00419=364547
BC00420=351830
BC00421=351830
BC00422=351830
BC00423=351830
BC00424=351830
BC00425=351830
BC00426=351830
BC00427=382963
BC00428=382962
BC00429=382962
BC00430=382962
BC00431=382962
BC00432=382962
BC00433=382962
BC00434=440664
BC00435=440664
BC00436=530314
BC00437=499273
BC00438=478480
BC00439=435223
BC00440=466651
BC00441=500323
BC00442=410824
BC00443=384863
BC00444=384863
BC00445=384863
BC00446=384863
BC00447=384863
BC00448=384863
BC00449=384863
BC00450=384863
BC00451=384246
BC00452=384246
BC00453=384246
BC00454=384246
BC00455=384246
BC00456=384246
BC00457=434425
BC00458=382279
BC00459=364547
BC00460=368602
BC00461=368602
BC00462=368602
BC00463=368602
BC00464=368602
BC00465=425990
BC00466=424496
BC00467=424496
BC00468=424496
BC00469=424496
BC00470=424496
BC00471=487434
BC00472=491487
BC00473=491487
BC00474=491487
BC00475=491487
BC00476=491487
BC00477=548878
BC00478=548005
BC00479=548005
BC00480=548005
BC00481=548005
BC00482=548005
BC00483=610322
BC00484=615349
BC00485=615349
BC00486=615349
BC00487=615349
BC00488=615349
BC00489=671766
BC00490=668615
BC00491=668615
BC00492=668615
BC00493=668615
BC00494=668615
BC00495=733216
BC00496=736931
BC00497=736931
BC00498=736931
BC00499=736931
BC00500=736931
BC00501=794661
BC00502=793324
BC00503=793324
BC00504=793324
BC00505=793324
BC00506=793324
BC00507=856105
BC00508=859171
BC00509=859171
BC00510=859171
BC00511=859171
BC00512=859171
BC00513=917549
BC00514=915489
BC00515=915489
BC00516=915489
BC00517=915489
BC00518=915489
BC00519=888684
BC00520=888684
BC00521=888684
BC00522=888684
BC00523=888684
BC00524=888684
BC00525=888684
BC00526=888684
BC00527=888684
BC00528=854699
BC00529=739244
BC00530=739244
BC00531=643789
BC00532=695024
BC00533=736803
BC00534=736803
BC00535=736800
BC00536=796843
BC00537=797249
BC00538=797249
BC00539=797249
BC00540=797249
BC00541=784304
BC00542=733836
BC00543=733836
BC00544=733836
BC00545=793674
BC00546=774393
BC00547=642838
BC00548=761950
BC00549=761950
BC00550=871390
BC00551=871390
BC00552=863896
BC00553=890558
BC00554=873393
BC00555=879870
BC00556=879870
BC00557=879870
BC00558=873394
BC00559=715867
BC00560=761950
BC00561=761950
BC00562=856724
BC00563=879459
BC00564=879459
BC00565=884890
BC00566=880213
BC00567=903175
BC00568=896757
BC00569=896245
BC00570=894993
BC00571=895155
BC00572=879459
BC00573=879459
BC00574=810641
BC00575=808033
BC00576=808033
BC00577=715610
BC00578=561575
BC00579=561575
BC00580=561572
BC00581=561572
BC00582=422137
BC00583=422137
BC00584=367622
BC00585=361480
BC00586=421627
BC00587=421627
BC00588=506917
BC00589=561572
BC00590=561575
BC00591=561575
BC00592=522965
BC00593=426143
BC00594=445051
BC00595=390808
BC00596=365835
BC00597=365835
BC00598=424019
BC00599=424019
BC00600=522965
BC00601=561575
BC00602=561575
BC00603=532118
BC00604=607170
BC00605=607170
BC00606=607170
BC00607=606544
BC00608=665714
BC00609=665899
BC00610=665899
BC00611=599364
BC00612=531162
BC00613=535379
BC00614=535379
BC00615=605958
BC00616=608441
BC00617=608441
BC00618=608441
BC00619=667817
BC00620=667920
BC00621=610149
BC00622=449249
BC00623=561572
BC00624=845683
BC00625=845683
BC00626=845683
BC00627=888208
BC00628=905757
BC00629=814209
BC00630=814209
BC00631=814209
BC00632=814209
BC00633=847657
BC00634=860371
BC00635=860371
BC00636=906357
BC00637=897737
BC00638=834201
BC00639=764098
BC00640=755906
BC00641=542328
BC00642=349973
BC00643=349973
BC00644=349973
BC00645=365825
BC00646=365825
BC00647=374698
BC00648=374698
BC00649=374698
BC00650=375082
BC00651=359453
BC00652=359342
BC00653=359337
BC00654=359337
BC00655=359337
BC00656=359337
BC00657=358620
BC00658=365825
BC00659=349973
BC00660=349973
BC00661=349973
BC00662=349974
BC00663=485414
BC00664=516640
BC00665=349973
BC00666=349971
BC00667=364871
BC00668=381296
BC00669=381296
BC00670=381295
BC00671=348430
BC00672=348430
BC00673=348430
BC00674=365935
BC00675=349510
BC00676=334610
BC00677=334612
BC00678=349973
BC00679=528150
BC00680=532118
BC00681=541988
BC00682=482330
BC00683=482330
BC00684=482330
BC00685=540008
BC00686=541106
BC00687=541106
BC00688=541106
BC00689=541106
BC00690=489272
BC00691=489272
BC00692=489272
BC00693=548185
BC00694=549104
BC00695=541106
BC00696=541106
BC00697=541108
///POSTYPE BASE
///RECTAN
///RCONF 1,0,0,0,0,0,0,0,0,0,0,0,0,0,0,0,0,0,0,0,0,0,0,0
P00006=0.000,0.000,0.000,0.0000,0.0000,0.0000
///RCONF 0,0,0,0,0,0,0,0,0,0,0,0,0,0,0,0,0,0,0,0,0,0,0,0
P00057=0.000,0.000,2.000,0.0000,0.0000,0.0000
P00058=0.000,0.000,3.000,0.0000,0.0000,0.0000
///RCONF 1,0,0,0,0,0,0,0,0,0,0,0,0,0,0,0,0,0,0,0,0,0,0,0
P00097=0.043,-1.896,1.568,0.0000,0.0000,0.0000
P00098=-0.089,-2.467,4.059,0.0000,0.0000,0.0000
P00099=0.011,-2.380,1.226,0.0000,0.0000,0.0000
P00100=-0.081,2.558,4.482,0.0000,0.0000,0.0000
P00101=0.030,-2.286,2.993,0.0000,0.0000,0.0000
P00102=-0.005,-1.108,1.644,0.0000,0.0000,0.0000
P00103=-0.094,-3.400,4.200,0.0000,0.0000,0.0000
P00104=0.043,-2.127,5.826,0.0000,0.0000,0.0000
P00105=-0.043,0.662,5.286,0.0000,0.0000,0.0000
P00106=-0.018,-2.519,0.237,0.0000,0.0000,0.0000
P00107=-0.008,-4.537,-4.500,0.0000,0.0000,0.0000
P00108=0.014,-3.040,2.637,0.0000,0.0000,0.0000
///RCONF 0,0,0,0,0,0,0,0,0,0,0,0,0,0,0,0,0,0,0,0,0,0,0,0
P00299=-1.404,-0.874,9.133,0.0000,0.0000,0.0000
///RCONF 1,0,0,0,0,0,0,0,0,0,0,0,0,0,0,0,0,0,0,0,0,0,0,0
P00301=0.046,-2.112,7.779,0.0000,0.0000,0.0000
P00302=-0.180,-2.409,6.326,0.0000,0.0000,0.0000
///RCONF 0,0,0,0,0,0,0,0,0,0,0,0,0,0,0,0,0,0,0,0,0,0,0,0
P00303=-0.004,-1.437,-4.584,0.0000,0.0000,0.0000
P00304=0.028,-1.666,-4.234,0.0000,0.0000,0.0000
P00305=-0.003,-1.920,-3.501,0.0000,0.0000,0.0000
P00306=0.015,-2.252,-3.054,0.0000,0.0000,0.0000
P00307=0.019,-2.151,-5.077,0.0000,0.0000,0.0000
P00308=-0.003,-2.092,-4.888,0.0000,0.0000,0.0000
P00309=-0.040,-2.205,-4.992,0.0000,0.0000,0.0000
P00310=-0.006,-2.490,-5.925,0.0000,0.0000,0.0000
P00311=-0.007,-2.079,-5.307,0.0000,0.0000,0.0000
P00312=-0.032,2.202,-7.632,0.0000,0.0000,0.0000
///RCONF 1,0,0,0,0,0,0,0,0,0,0,0,0,0,0,0,0,0,0,0,0,0,0,0
P00349=0.060,0.167,-1.133,0.0000,0.0000,0.0000
///RCONF 0,0,0,0,0,0,0,0,0,0,0,0,0,0,0,0,0,0,0,0,0,0,0,0
P00350=11.519,-0.008,1.149,0.0000,0.0000,0.0000
P00351=13.563,-0.027,-0.653,0.0000,0.0000,0.0000
P00352=13.252,-0.027,-0.827,0.0000,0.0000,0.0000
P00353=10.971,-0.082,0.776,0.0000,0.0000,0.0000
P00354=-0.024,2.508,-1.824,0.0000,0.0000,0.0000
P00355=-0.001,2.528,-1.131,0.0000,0.0000,0.0000
P00356=-0.034,2.921,-0.262,0.0000,0.0000,0.0000
P00357=0.003,3.386,-0.091,0.0000,0.0000,0.0000
P00358=0.014,3.037,-0.020,0.0000,0.0000,0.0000
P00359=-0.005,2.731,0.912,0.0000,0.0000,0.0000
P00360=-0.011,3.412,0.438,0.0000,0.0000,0.0000
P00361=0.018,3.050,1.253,0.0000,0.0000,0.0000
P00399=-2.449,0.031,8.825,0.0000,0.0000,0.0000
P00400=5.920,-3.503,-0.024,0.0000,0.0000,0.0000
P00401=3.430,-0.021,1.131,0.0000,0.0000,0.0000
P00402=-0.253,1.107,3.062,0.0000,0.0000,0.0000
P00403=-3.666,-0.015,5.328,0.0000,0.0000,0.0000
P00405=2.420,0.007,1.427,0.0000,0.0000,0.0000
P00406=3.513,-0.022,0.429,0.0000,0.0000,0.0000
P00415=-1.781,-1.303,3.250,0.0000,0.0000,0.0000
P00416=0.027,1.119,3.078,0.0000,0.0000,0.0000
//INST
///DATE 2025/02/05 14:43
///ATTR SC,RW
///GROUP1 RB1,BS1
NOP
CALL JOB:MOVE_INTO_TUNNEL
SFTOF
'------------------------
'------------------------
'SPOINA SRODEK DOL
'------------------------
'------------------------
MOVJ C00000 BC00000 VJ=10.00
MOVJ C00001 BC00001 VJ=30.00
'------------------------
'PODLOGA_BEZ_ROZPORKI
'------------------------
'TEST
MOVL C00002 BC00002 V=166.7
MOVL C00003 BC00003 V=166.7 PL=0
REFP 3 C00004 BC00004
CALL JOB:SEARCH-R1
IMOV P0057 V=23.0
SET P0097 P0006
SFTON P0097
REFP 3 C00005 BC00005
CALL JOB:SEARCH-R1
SET P0097 P0006
SFTON P0097
MOVL C00006 BC00006 V=166.7 PL=0
SFTOF
COMM MOVL C00007 BC00007 V=333.3
MOVL C00008 BC00008 V=333.3
MOVL C00009 BC00009 V=166.7 PL=0
REFP 3 C00010 BC00010
CALL JOB:SEARCH-R1
IMOV P0057 V=23.0
SET P0098 P0006
SFTON P0098
REFP 3 C00011 BC00011
CALL JOB:SEARCH-R1
SET P0098 P0006
SFTON P0098
MOVL C00012 BC00012 V=166.7 PL=0
'TEST
SFTOF
'------------------------
'W38 P
'------------------------
'TEST
MOVL C00013 BC00013 V=166.7
MOVL C00014 BC00014 V=166.7 PL=0
REFP 3 C00015 BC00015
CALL JOB:SEARCH-R1
IMOV P0057 V=23.0
SET P0099 P0006
SFTON P0099
REFP 3 C00016 BC00016
CALL JOB:SEARCH-R1
SET P0099 P0006
SFTON P0099
MOVL C00017 BC00017 V=166.7 PL=0
'TEST
SFTOF
MOVL C00018 BC00018 V=333.3
MOVL C00019 BC00019 V=333.3
'------------------------
'W38 L
'------------------------
'TEST
MOVL C00020 BC00020 V=166.7 PL=0
REFP 3 C00021 BC00021
CALL JOB:SEARCH-R1
IMOV P0057 V=23.0
SET P0100 P0006
SFTON P0100
REFP 3 C00022 BC00022
CALL JOB:SEARCH-R1
SET P0100 P0006
SFTON P0100
MOVL C00023 BC00023 V=166.7 PL=0
'TEST
SFTOF
MOVJ C00024 BC00024 VJ=20.00
'------------------------
'W45 P
'------------------------
MOVL C00025 BC00025 V=166.7 PL=0
REFP 3 C00026 BC00026
CALL JOB:SEARCH-R1
IMOV P0057 V=23.0
SET P0101 P0006
SFTON P0101
REFP 3 C00027 BC00027
CALL JOB:SEARCH-R1
SET P0101 P0006
SFTON P0101
MOVL C00028 BC00028 V=166.7 PL=0
'TEST
SFTOF
MOVJ C00029 BC00029 VJ=20.00
'------------------------
'W45 L
'------------------------
MOVL C00030 BC00030 V=133.3 PL=0
REFP 3 C00031 BC00031
CALL JOB:SEARCH-R1
IMOV P0057 V=23.0
SET P0102 P0006
SFTON P0102
REFP 3 C00032 BC00032
CALL JOB:SEARCH-R1
SET P0102 P0006
SFTON P0102
MOVL C00033 BC00033 V=250.0 PL=0
'TEST
SFTOF
MOVJ C00034 BC00034 VJ=30.00
MOVJ C00035 BC00035 VJ=30.00
MOVJ C00036 BC00036 VJ=20.00
'------------------------
'W48 P
'------------------------
'TEST
MOVL C00037 BC00037 V=133.3 PL=0
REFP 3 C00038 BC00038
CALL JOB:SEARCH-R1
IMOV P0057 V=23.0
SET P0103 P0006
SFTON P0103
REFP 3 C00039 BC00039
CALL JOB:SEARCH-R1
SET P0103 P0006
SFTON P0103
MOVL C00040 BC00040 V=166.7 PL=0
'TEST
SFTOF
COMM MOVJ C00041 BC00041 VJ=30.00
COMM MOVJ C00042 BC00042 VJ=30.00
COMM MOVJ C00043 BC00043 VJ=30.00
COMM MOVJ C00044 BC00044 VJ=30.00
COMM MOVJ C00045 BC00045 VJ=20.00
MOVL C00046 BC00046 V=250.0
'------------------------
'W48 L
'------------------------
SFTOF
MOVL C00047 BC00047 V=133.3 PL=0
REFP 3 C00048 BC00048
CALL JOB:SEARCH-R1
IMOV P0057 V=23.0
SET P0104 P0006
SFTON P0104
REFP 3 C00049 BC00049
CALL JOB:SEARCH-R1
SET P0104 P0006
SFTON P0104
MOVL C00050 BC00050 V=166.7 PL=0
SFTOF
MOVJ C00051 BC00051 VJ=20.00
'------------------------
'W36 P
'------------------------
MOVL C00052 BC00052 V=133.3 PL=0
REFP 3 C00053 BC00053
CALL JOB:SEARCH-R1
IMOV P0057 V=23.0
SET P0105 P0006
SFTON P0105
REFP 3 C00054 BC00054
CALL JOB:SEARCH-R1
SET P0105 P0006
SFTON P0105
MOVL C00055 BC00055 V=166.7 PL=0
'TEST
SFTOF
MOVJ C00056 BC00056 VJ=20.00
'------------------------
'W36 L
'------------------------
MOVL C00057 BC00057 V=166.7 PL=0
REFP 3 C00058 BC00058
CALL JOB:SEARCH-R1
IMOV P0057 V=23.0
SET P0106 P0006
SFTON P0106
REFP 3 C00059 BC00059
CALL JOB:SEARCH-R1
SET P0106 P0006
SFTON P0106
SFTOF
MOVL C00060 BC00060 V=166.7 PL=0
MOVJ C00061 BC00061 VJ=25.00
MOVJ C00062 BC00062 VJ=25.00
'TEST
MOVJ C00063 BC00063 VJ=20.00
SFTOF
'------------------------
'W44 P
'------------------------
'TEST
MOVL C00064 BC00064 V=133.3 PL=0
REFP 3 C00065 BC00065
CALL JOB:SEARCH-R1
IMOV P0057 V=23.0
SET P0107 P0006
SFTON P0107
REFP 3 C00066 BC00066
CALL JOB:SEARCH-R1
SET P0107 P0006
SFTON P0107
SFTOF
MOVL C00067 BC00067 V=250.0 PL=0
'TEST
MOVL C00068 BC00068 V=416.7
MOVL C00069 BC00069 V=166.7 PL=0
REFP 3 C00070 BC00070
CALL JOB:SEARCH-R1
IMOV P0057 V=23.0
SET P0108 P0006
SFTON P0108
REFP 3 C00071 BC00071
CALL JOB:SEARCH-R1
SET P0108 P0006
SFTON P0108
SFTOF
MOVL C00072 BC00072 V=250.0 PL=0
'TEST
SFTOF
MOVL C00073 BC00073 V=250.0
MOVJ C00074 BC00074 VJ=25.00
CALL JOB:FRONT_SEARCH_0ST-2_4740
COMM MOVJ C00075 BC00075 VJ=20.00
COMM MOVJ C00076 BC00076 VJ=20.00
COMM MOVJ C00077 BC00077 VJ=20.00
COMM 'DODANE
COMM 'SZUKANIE FRONT
COMM '------------------------
COMM '503
COMM '------------------------
COMM MOVL C00078 BC00078 V=333.3
COMM MOVL C00079 BC00079 V=166.7 PL=0
COMM REFP 3 C00080 BC00080
COMM CALL JOB:SEARCH-R1
COMM IMOV P0058 V=16.7
COMM SET P0350 P0006
COMM SFTON P0350
COMM REFP 3 C00081 BC00081
COMM CALL JOB:SEARCH-R1
COMM SET P0350 P0006
COMM SFTON P0350
COMM MOVL C00082 BC00082 V=66.7 PL=0
COMM SFTOF
COMM '------------------------
COMM '------------------------
COMM '502
COMM '------------------------
COMM MOVL C00083 BC00083 V=166.7
COMM MOVL C00084 BC00084 V=66.7 PL=0
COMM REFP 3 C00085 BC00085
COMM CALL JOB:SEARCH-R1
COMM IMOV P0058 V=16.7
COMM SET P0351 P0006
COMM SFTON P0351
COMM REFP 3 C00086 BC00086
COMM CALL JOB:SEARCH-R1
COMM SET P0351 P0006
COMM SFTON P0351
COMM MOVL C00087 BC00087 V=66.7 PL=0
COMM SFTOF
COMM '------------------------
COMM '------------------------
COMM '501
COMM '------------------------
COMM MOVL C00088 BC00088 V=166.7
COMM MOVL C00089 BC00089 V=66.7 PL=0
COMM REFP 3 C00090 BC00090
COMM CALL JOB:SEARCH-R1
COMM IMOV P0058 V=16.7
COMM SET P0352 P0006
COMM SFTON P0352
COMM REFP 3 C00091 BC00091
COMM CALL JOB:SEARCH-R1
COMM SET P0352 P0006
COMM SFTON P0352
COMM MOVL C00092 BC00092 V=66.7 PL=0
COMM SFTOF
COMM '------------------------
COMM '------------------------
COMM '500
COMM '------------------------
COMM MOVL C00093 BC00093 V=166.7
COMM MOVL C00094 BC00094 V=66.7 PL=0
COMM REFP 3 C00095 BC00095
COMM CALL JOB:SEARCH-R1
COMM IMOV P0058 V=16.7
COMM SET P0353 P0006
COMM SFTON P0353
COMM REFP 3 C00096 BC00096
COMM CALL JOB:SEARCH-R1
COMM SET P0353 P0006
COMM SFTON P0353
COMM MOVL C00097 BC00097 V=66.7 PL=0
COMM SFTOF
COMM '------------------------
COMM MOVL C00098 BC00098 V=333.3
COMM MOVL C00099 BC00099 V=333.3
COMM MOVJ C00100 BC00100 VJ=10.00
COMM 'DODANE
COMM MOVJ C00101 BC00101 VJ=10.00
COMM '------------------------
COMM 'SFT402
COMM '------------------------
COMM SFTOF
COMM MOVL C00102 BC00102 V=150.0
COMM MOVL C00103 BC00103 V=66.7 PL=0
COMM REFP 3 C00104 BC00104
COMM CALL JOB:SEARCH-R1
COMM SET P0402 P0006
COMM SFTON P0402
COMM MOVL C00105 BC00105 V=150.0
COMM MOVL C00106 BC00106 V=66.7 PL=0
COMM REFP 3 C00107 BC00107
COMM CALL JOB:SEARCH-R1
COMM SET P0402 P0006
COMM SFTON P0402
COMM MOVL C00108 BC00108 V=133.3
COMM MOVL C00109 BC00109 V=150.0
COMM MOVL C00110 BC00110 V=150.0
COMM MOVL C00111 BC00111 V=66.7 PL=0
COMM REFP 3 C00112 BC00112
COMM CALL JOB:SEARCH-R1
COMM SET P0402 P0006
COMM SFTOF
COMM MOVL C00113 BC00113 V=150.0
COMM '------------------------
COMM 'SFT403
COMM '------------------------
COMM 'START
COMM SFTOF
COMM MOVL C00114 BC00114 V=250.0
COMM MOVL C00115 BC00115 V=133.3 PL=0
COMM REFP 3 C00116 BC00116
COMM CALL JOB:SEARCH-R1
COMM SET P0416 P0006
COMM SFTON P0416
COMM MOVL C00117 BC00117 V=133.3
COMM REFP 3 C00118 BC00118
COMM CALL JOB:SEARCH-R1
COMM SET P0402 P0006
COMM SFTOF
COMM MOVL C00119 BC00119 V=150.0
COMM '------------------------
COMM '------------------------
COMM SFTOF
COMM MOVL C00120 BC00120 V=250.0
COMM MOVL C00121 BC00121 V=133.3 PL=0
COMM REFP 3 C00122 BC00122
COMM CALL JOB:SEARCH-R1
COMM SET P0403 P0006
COMM SFTON P0403
COMM MOVL C00123 BC00123 V=66.7 PL=0
COMM REFP 3 C00124 BC00124
COMM CALL JOB:SEARCH-R1
COMM SET P0403 P0006
COMM SFTOF
COMM MOVL C00125 BC00125 V=150.0
COMM MOVJ C00126 BC00126 VJ=20.00
COMM MOVJ C00127 BC00127 VJ=20.00
COMM '------------------------
COMM 'SFT401
COMM '------------------------
COMM SFTOF
COMM MOVL C00128 BC00128 V=150.0
COMM MOVL C00129 BC00129 V=66.7 PL=0
COMM REFP 3 C00130 BC00130
COMM CALL JOB:SEARCH-R1
COMM SET P0401 P0006
COMM SFTON P0401
COMM MOVL C00131 BC00131 V=66.7 PL=0
COMM REFP 3 C00132 BC00132
COMM CALL JOB:SEARCH-R1
COMM SET P0401 P0006
COMM SFTOF
COMM MOVL C00133 BC00133 V=150.0
COMM 'SFT400
COMM '------------------------
COMM SFTOF
COMM MOVL C00134 BC00134 V=333.3
COMM MOVL C00135 BC00135 V=66.7 PL=0
COMM REFP 3 C00136 BC00136
COMM CALL JOB:SEARCH-R1
COMM SET P0405 P0006
COMM SFTON P0405
COMM MOVL C00137 BC00137 V=66.7 PL=0
COMM REFP 3 C00138 BC00138
COMM CALL JOB:SEARCH-R1
COMM SET P0405 P0006
COMM SFTOF
COMM MOVL C00139 BC00139 V=150.0
COMM 'SFT400
COMM '------------------------
COMM SFTOF
COMM MOVL C00140 BC00140 V=333.3
COMM MOVL C00141 BC00141 V=133.3 PL=0
COMM REFP 3 C00142 BC00142
COMM CALL JOB:SEARCH-R1
COMM SET P0406 P0006
COMM SFTON P0406
COMM MOVL C00143 BC00143 V=66.7 PL=0
COMM REFP 3 C00144 BC00144
COMM CALL JOB:SEARCH-R1
COMM SET P0406 P0006
COMM SFTOF
COMM MOVL C00145 BC00145 V=150.0
COMM 'SFT400
COMM '------------------------
COMM SFTOF
COMM MOVL C00146 BC00146 V=150.0
COMM MOVL C00147 BC00147 V=66.7 PL=0
COMM REFP 3 C00148 BC00148
COMM CALL JOB:SEARCH-R1
COMM SET P0400 P0006
COMM SFTON P0400
COMM MOVL C00149 BC00149 V=150.0
COMM MOVL C00150 BC00150 V=66.7 PL=0
COMM REFP 3 C00151 BC00151
COMM CALL JOB:SEARCH-R1
COMM SET P0400 P0006
COMM SFTON P0400
COMM MOVL C00152 BC00152 V=150.0
COMM MOVL C00153 BC00153 V=150.0
COMM MOVL C00154 BC00154 V=66.7 PL=0
COMM REFP 3 C00155 BC00155
COMM CALL JOB:SEARCH-R1
COMM SET P0400 P0006
COMM SFTOF
COMM MOVL C00156 BC00156 V=83.3
COMM MOVL C00157 BC00157 V=250.0
COMM MOVL C00158 BC00158 V=333.3
COMM MOVL C00159 BC00159 V=66.7 PL=0
COMM REFP 3 C00160 BC00160
COMM CALL JOB:SEARCH-R1
COMM SET P0415 P0006
COMM SFTON P0415
COMM MOVL C00161 BC00161 V=133.3
COMM REFP 3 C00162 BC00162
COMM CALL JOB:SEARCH-R1
COMM SET P0415 P0006
COMM SFTOF
COMM MOVL C00163 BC00163 V=150.0
COMM '------------------------
COMM 'SFT403
COMM '------------------------
COMM 'START
COMM SFTOF
COMM MOVJ C00164 BC00164 VJ=10.00
COMM '------------------------
COMM 'SFT399
COMM '------------------------
COMM 'START
COMM SFTOF
COMM MOVL C00165 BC00165 V=150.0
COMM MOVL C00166 BC00166 V=66.7 PL=0
COMM REFP 3 C00167 BC00167
COMM CALL JOB:SEARCH-R1
COMM SET P0399 P0006
COMM SFTON P0399
COMM MOVL C00168 BC00168 V=66.7 PL=0
COMM REFP 3 C00169 BC00169
COMM CALL JOB:SEARCH-R1
COMM SET P0399 P0006
COMM SFTOF
COMM MOVL C00170 BC00170 V=150.0
COMM MOVJ C00171 BC00171 VJ=20.00
COMM MOVJ C00172 BC00172 VJ=30.00
COMM MOVJ C00173 BC00173 VJ=30.00
COMM MOVJ C00174 BC00174 VJ=30.00
MOVJ C00175 BC00175 VJ=40.00
'WELD
'WELD
MOVJ C00176 BC00176 VJ=20.00
'**********************
'W36
'**********************
MOVL C00177 BC00177 V=500.0
SFTON P0105
MOVL C00178 BC00178 V=166.7 PL=0
SFTOF
MACRO1 MJ#(0) ARGF24
ARCON
SFTON P0106
MOVL C00179 BC00179 V=11.0
ARCOF
SFTOF
MOVJ C00180 BC00180 VJ=15.00
MOVJ C00181 BC00181 VJ=30.00
MOVJ C00182 BC00182 VJ=10.00
MOVJ C00183 BC00183 VJ=10.00
MOVJ C00184 BC00184 VJ=30.00
MOVJ C00185 BC00185 VJ=20.00
MOVJ C00186 BC00186 VJ=10.00
MOVJ C00187 BC00187 VJ=15.00
'**********************
'W38
'**********************
MOVL C00188 BC00188 V=500.0
SFTON P0100
MOVL C00189 BC00189 V=166.7 PL=0
SFTOF
ARCON
SFTON P0099
MOVL C00190 BC00190 V=11.0
ARCOF
SFTOF
'DODANE
MOVL C00191 BC00191 V=500.0
MOVL C00192 BC00192 V=666.7
MOVJ C00193 BC00193 VJ=10.00
MOVJ C00194 BC00194 VJ=10.00
MOVJ C00195 BC00195 VJ=10.00
MOVJ C00196 BC00196 VJ=10.00
MOVJ C00197 BC00197 VJ=25.00
COMM '**********************
COMM '**********************
COMM 'POCZATEK SPAWANIA PRZOD
COMM '**********************
COMM '**********************
COMM MOVJ C00198 BC00198 VJ=30.00
COMM MOVL C00199 BC00199 V=416.7
COMM MOVJ C00200 BC00200 VJ=10.00
COMM MOVJ C00201 BC00201 VJ=10.00
COMM MOVL C00202 BC00202 V=150.0
COMM MOVL C00203 BC00203 V=150.0
COMM '**********************
COMM 'W41A SIDE
COMM '**********************
COMM MOVL C00204 BC00204 V=250.0
COMM SFTON P0402
COMM MOVL C00205 BC00205 V=66.7 PL=0
COMM MACRO1 MJ#(0) ARGF14
COMM ARCON
COMM MOVL C00206 BC00206 V=9.2
COMM ARCOF
COMM SFTOF
COMM MOVL C00207 BC00207 V=166.7
COMM '**********************
COMM 'W41A FRONT
COMM '**********************
COMM MOVL C00208 BC00208 V=250.0
COMM SFTON P0350
COMM MOVL C00209 BC00209 V=66.7 PL=0
COMM SFTOF
COMM MACRO1 MJ#(0) ARGF21
COMM ARCON
COMM SFTON P0351
COMM MOVL C00210 BC00210 V=8.3
COMM SFTOF
COMM ARCOF
COMM MOVL C00211 BC00211 V=166.7
COMM '**********************
COMM 'W41B FRONT
COMM '**********************
COMM MOVL C00212 BC00212 V=250.0
COMM SFTON P0352
COMM MOVL C00213 BC00213 V=66.7 PL=0
COMM SFTOF
COMM MACRO1 MJ#(0) ARGF21
COMM ARCON
COMM SFTON P0353
COMM MOVL C00214 BC00214 V=8.3
COMM SFTOF
COMM ARCOF
COMM MOVL C00215 BC00215 V=166.7
COMM MOVL C00216 BC00216 V=100.0
COMM '**********************
COMM 'W41A SIDE
COMM '**********************
COMM SFTON P0400
COMM MOVL C00217 BC00217 V=66.7 PL=0
COMM MACRO1 MJ#(0) ARGF21
COMM ARCON
COMM MOVL C00218 BC00218 V=8.3
COMM ARCOF
COMM SFTOF
COMM MOVL C00219 BC00219 V=166.7
COMM MOVL C00220 BC00220 V=166.7
COMM MOVL C00221 BC00221 V=333.3
COMM MOVJ C00222 BC00222 VJ=20.00
COMM MOVJ C00223 BC00223 VJ=20.00
COMM '**********************
COMM 'W42A.1
COMM '**********************
COMM 'POPRAWIC
COMM MOVL C00224 BC00224 V=500.0
COMM SFTON P0403
COMM MOVL C00225 BC00225 V=66.7 PL=0
COMM MACRO1 MJ#(0) ARGF9
COMM ARCON
COMM MOVL C00226 BC00226 V=9.2
COMM SFTON P0416
COMM MOVL C00227 BC00227 V=9.2
COMM MOVL C00228 BC00228 V=9.2
COMM MOVL C00229 BC00229 V=9.2
COMM SFTON P0402
COMM MOVL C00230 BC00230 V=9.2
COMM MOVL C00231 BC00231 V=9.2
COMM ARCOF
COMM MOVL C00232 BC00232 V=500.0
COMM SFTOF
COMM MOVJ C00233 BC00233 VJ=15.00
COMM 'W42B.1
COMM MOVJ C00234 BC00234 VJ=30.00
COMM MOVJ C00235 BC00235 VJ=30.00
COMM MOVJ C00236 BC00236 VJ=30.00
COMM MOVJ C00237 BC00237 VJ=30.00
COMM '**********************
COMM 'W42B.1
COMM '**********************
COMM MOVL C00238 BC00238 V=500.0
COMM SFTON P0399
COMM MOVL C00239 BC00239 V=66.7 PL=0
COMM MACRO1 MJ#(0) ARGF9
COMM ARCON
COMM SFTON P0415
COMM MOVL C00240 BC00240 V=9.2
COMM MOVL C00241 BC00241 V=9.2
COMM MOVL C00242 BC00242 V=9.2
COMM SFTON P0400
COMM MOVL C00243 BC00243 V=9.2
COMM MOVL C00244 BC00244 V=9.2
COMM ARCOF
COMM MOVL C00245 BC00245 V=500.0
COMM SFTOF
COMM MOVJ C00246 BC00246 VJ=15.00
COMM 'W42A.2
COMM MOVJ C00247 BC00247 VJ=20.00
COMM MOVJ C00248 BC00248 VJ=20.00
COMM MOVJ C00249 BC00249 VJ=20.00
COMM MOVJ C00250 BC00250 VJ=20.00
COMM MOVJ C00251 BC00251 VJ=20.00
COMM '**********************
COMM 'W42A.2
COMM '**********************
COMM MOVL C00252 BC00252 V=500.0
COMM SFTON P0402
COMM MOVL C00253 BC00253 V=66.7 PL=0
COMM SFTOF
COMM MACRO1 MJ#(0) ARGF9
COMM ARCON
COMM SFTON P0402
COMM MOVL C00254 BC00254 V=9.2
COMM ARCOF
COMM MOVL C00255 BC00255 V=166.7
COMM MOVJ C00256 BC00256 VJ=20.00
COMM MOVJ C00257 BC00257 VJ=20.00
COMM MOVL C00258 BC00258 V=166.7
COMM MOVL C00259 BC00259 V=166.7
COMM ARCON
COMM MOVL C00260 BC00260 V=10.8
COMM ARCOF
COMM MOVL C00261 BC00261 V=166.7
COMM MOVJ C00262 BC00262 VJ=10.00
COMM SFTOF
COMM MOVJ C00263 BC00263 VJ=20.00
COMM MOVJ C00264 BC00264 VJ=20.00
COMM MOVJ C00265 BC00265 VJ=20.00
COMM 'W42B.2
COMM MOVJ C00266 BC00266 VJ=20.00
COMM MOVJ C00267 BC00267 VJ=20.00
COMM MOVJ C00268 BC00268 VJ=20.00
COMM MOVJ C00269 BC00269 VJ=20.00
COMM MOVJ C00270 BC00270 VJ=20.00
COMM '**********************
COMM 'W42B.2
COMM '**********************
COMM MOVL C00271 BC00271 V=500.0
COMM SFTON P0400
COMM MOVL C00272 BC00272 V=166.7 PL=0
COMM SFTOF
COMM MACRO1 MJ#(0) ARGF9
COMM ARCON
COMM SFTON P0400
COMM MOVL C00273 BC00273 V=9.2
COMM ARCOF
COMM SFTOF
COMM MOVL C00274 BC00274 V=166.7
COMM MOVL C00275 BC00275 V=166.7
COMM MOVJ C00276 BC00276 VJ=10.00
COMM SFTON P0400
COMM MOVL C00277 BC00277 V=166.7
COMM ARCON
COMM MOVL C00278 BC00278 V=10.8
COMM ARCOF
COMM MOVL C00279 BC00279 V=166.7
COMM MOVL C00280 BC00280 V=500.0
COMM SFTOF
COMM MOVJ C00281 BC00281 VJ=20.00
COMM MOVJ C00282 BC00282 VJ=20.00
COMM 'W42A.3
COMM MOVJ C00283 BC00283 VJ=10.00
COMM MOVJ C00284 BC00284 VJ=20.00
COMM MOVJ C00285 BC00285 VJ=20.00
COMM MOVJ C00286 BC00286 VJ=20.00
COMM '**********************
COMM 'W42A.3
COMM '**********************
COMM MOVL C00287 BC00287 V=500.0
COMM SFTON P0402
COMM MOVL C00288 BC00288 V=166.7 PL=0
COMM MACRO1 MJ#(0) ARGF9
COMM ARCON
COMM MOVL C00289 BC00289 V=9.2
COMM ARCOF
COMM MOVL C00290 BC00290 V=500.0
COMM SFTOF
COMM '**********************
COMM 'W42B.3
COMM '**********************
COMM MOVL C00291 BC00291 V=500.0
COMM SFTON P0400
COMM MOVL C00292 BC00292 V=66.7 PL=0
COMM ARCON
COMM MOVL C00293 BC00293 V=9.2
COMM ARCOF
COMM MOVL C00294 BC00294 V=500.0
COMM SFTOF
COMM MOVJ C00295 BC00295 VJ=10.00
COMM '**********************
COMM 'GORA L
COMM '**********************
COMM MOVL C00296 BC00296 V=500.0
COMM SFTON P0401
COMM MOVL C00297 BC00297 V=66.7 PL=0
COMM MACRO1 MJ#(0) ARGF9
COMM ARCON
COMM MOVL C00298 BC00298 V=11.7
COMM SFTON P0406
COMM MOVL C00299 BC00299 V=11.7
COMM MOVL C00300 BC00300 V=11.7
COMM MOVL C00301 BC00301 V=11.7
COMM ARCOF
COMM MOVL C00302 BC00302 V=500.0
COMM SFTOF
COMM '**********************
COMM 'GORA P
COMM '**********************
COMM MOVL C00303 BC00303 V=166.7
COMM SFTON P0401
COMM MOVL C00304 BC00304 V=166.7 PL=0
COMM ARCON
COMM MOVL C00305 BC00305 V=11.7
COMM SFTON P0405
COMM MOVL C00306 BC00306 V=11.7
COMM MOVL C00307 BC00307 V=11.7
COMM MOVL C00308 BC00308 V=11.7
COMM ARCOF
COMM MOVL C00309 BC00309 V=500.0
COMM SFTOF
COMM MOVJ C00310 BC00310 VJ=10.00
COMM MOVJ C00311 BC00311 VJ=30.00
COMM MOVJ C00312 BC00312 VJ=30.00
COMM 'KONIEC SPAWANIA FRONTU
COMM '**********************
COMM 'W44
COMM '**********************
MOVJ C00313 BC00313 VJ=30.00
MOVJ C00314 BC00314 VJ=25.00
MOVJ C00315 BC00315 VJ=30.00
MOVJ C00316 BC00316 VJ=30.00
MOVL C00317 BC00317 V=500.0
SFTON P0108
MOVL C00318 BC00318 V=166.7 PL=0
MACRO1 MJ#(0) ARGF24
ARCON
MOVL C00319 BC00319 V=10.8
SFTON P0107
MOVL C00320 BC00320 V=10.8
MOVL C00321 BC00321 V=10.8
ARCOF
SFTOF
MOVL C00322 BC00322 V=500.0
MOVL C00323 BC00323 V=500.0
MOVJ C00324 BC00324 VJ=30.00
'**********************
'W45
'**********************
MOVJ C00325 BC00325 VJ=30.00
MOVJ C00326 BC00326 VJ=20.00
MOVJ C00327 BC00327 VJ=10.00
MACRO1 MJ#(0) ARGF24
MOVL C00328 BC00328 V=500.0
SFTON P0102
MOVL C00329 BC00329 V=166.7 PL=0
ARCON
SFTON P0101
MOVL C00330 BC00330 V=12.5
ARCOF
SFTOF
MOVL C00331 BC00331 V=500.0
'**********************
'SPOINA_PODLOGA_BRAK_ROZP
'**********************
MOVL C00332 BC00332 V=500.0
MOVL C00333 BC00333 V=500.0
SFTON P0098
MOVL C00334 BC00334 V=166.7 PL=0
SFTOF
ARCON
SFTON P0097
MOVL C00335 BC00335 V=11.3
ARCOF
SFTOF
MOVL C00336 BC00336 V=166.7
'DODANE
MOVJ C00337 BC00337 VJ=10.00
'**********************
'W48
'**********************
MOVJ C00338 BC00338 VJ=15.00
MOVJ C00339 BC00339 VJ=25.00
MOVJ C00340 BC00340 VJ=15.00
SFTON P0104
MOVL C00341 BC00341 V=166.7 PL=0
SFTOF
ARCON
SFTON P0103
MOVL C00342 BC00342 V=10.5
ARCOF
SFTOF
MOVL C00343 BC00343 V=500.0
MOVJ C00344 BC00344 VJ=40.00
CALL JOB:FRONT_WELD_0ST-2_4740
CALL JOB:MOVE_OUT_OF_TUNNEL
CALL JOB:CLEAN-R1
CALL JOB:MOVE_INTO_TUNNEL
MOVJ C00345 BC00345 VJ=30.00 PL=0
'------------------------
'------------------------
'PRAWA STRONA PROFIL GORA
'------------------------
'------------------------
MOVJ C00346 BC00346 VJ=20.00
'------------------------
'W51A L
'------------------------
SFTOF
MOVJ C00347 BC00347 VJ=10.00
MOVL C00348 BC00348 V=66.7 PL=0
REFP 3 C00349 BC00349
CALL JOB:SEARCH-R1
SET P0299 P0006
SFTON P0299
MOVL C00350 BC00350 V=66.7 PL=0
REFP 3 C00351 BC00351
CALL JOB:SEARCH-R1
SET P0299 P0006
SFTON P0299
MOVL C00352 BC00352 V=83.3
MOVL C00353 BC00353 V=166.7 PL=0
REFP 3 C00354 BC00354
CALL JOB:SEARCH-R1
SET P0299 P0006
SFTON P0299
MOVL C00355 BC00355 V=133.3 PL=0
SFTOF
'------------------------
'W51A P
'------------------------
SFTOF
MOVL C00356 BC00356 V=250.0
'------------------------
'W54A L
'------------------------
SFTOF
MOVJ C00357 BC00357 VJ=30.00
MOVL C00358 BC00358 V=133.3 PL=0
REFP 3 C00359 BC00359
CALL JOB:SEARCH-R1
SET P0301 P0006
SFTON P0301
MOVL C00360 BC00360 V=66.7 PL=0
REFP 3 C00361 BC00361
CALL JOB:SEARCH-R1
SET P0301 P0006
SFTON P0301
MOVL C00362 BC00362 V=66.7 PL=0
SFTOF
'------------------------
'W54A P
'------------------------
SFTOF
MOVJ C00363 BC00363 VJ=30.00
MOVL C00364 BC00364 V=133.3 PL=0
REFP 3 C00365 BC00365
CALL JOB:SEARCH-R1
SET P0302 P0006
SFTON P0302
MOVL C00366 BC00366 V=66.7 PL=0
REFP 3 C00367 BC00367
CALL JOB:SEARCH-R1
SET P0302 P0006
SFTON P0302
MOVL C00368 BC00368 V=66.7 PL=0
SFTOF
'------------------------
'W50A L
'------------------------
SFTOF
MOVJ C00369 BC00369 VJ=30.00
MOVL C00370 BC00370 V=133.3 PL=0
REFP 3 C00371 BC00371
CALL JOB:SEARCH-R1
SET P0303 P0006
SFTON P0303
MOVL C00372 BC00372 V=66.7 PL=0
REFP 3 C00373 BC00373
CALL JOB:SEARCH-R1
SET P0303 P0006
SFTON P0303
MOVL C00374 BC00374 V=66.7 PL=0
SFTOF
'------------------------
'W50A P
'------------------------
SFTOF
MOVJ C00375 BC00375 VJ=30.00
MOVL C00376 BC00376 V=133.3 PL=0
REFP 3 C00377 BC00377
CALL JOB:SEARCH-R1
SET P0304 P0006
SFTON P0304
MOVL C00378 BC00378 V=66.7 PL=0
REFP 3 C00379 BC00379
CALL JOB:SEARCH-R1
SET P0304 P0006
SFTON P0304
MOVL C00380 BC00380 V=66.7 PL=0
SFTOF
'------------------------
'W53A L
'------------------------
SFTOF
MOVJ C00381 BC00381 VJ=30.00
MOVL C00382 BC00382 V=133.3 PL=0
REFP 3 C00383 BC00383
CALL JOB:SEARCH-R1
SET P0305 P0006
SFTON P0305
MOVL C00384 BC00384 V=66.7 PL=0
REFP 3 C00385 BC00385
CALL JOB:SEARCH-R1
SET P0305 P0006
SFTON P0305
MOVL C00386 BC00386 V=66.7 PL=0
SFTOF
'------------------------
'W53A P
'------------------------
SFTOF
MOVJ C00387 BC00387 VJ=30.00
MOVL C00388 BC00388 V=200.0
MOVL C00389 BC00389 V=66.7 PL=0
REFP 3 C00390 BC00390
CALL JOB:SEARCH-R1
SET P0306 P0006
SFTON P0306
MOVL C00391 BC00391 V=66.7 PL=0
REFP 3 C00392 BC00392
CALL JOB:SEARCH-R1
SET P0306 P0006
SFTON P0306
MOVL C00393 BC00393 V=66.7 PL=0
SFTOF
'------------------------
'W56A L
'------------------------
SFTOF
MOVJ C00394 BC00394 VJ=30.00
MOVL C00395 BC00395 V=133.3 PL=0
REFP 3 C00396 BC00396
CALL JOB:SEARCH-R1
SET P0307 P0006
SFTON P0307
MOVL C00397 BC00397 V=66.7 PL=0
REFP 3 C00398 BC00398
CALL JOB:SEARCH-R1
SET P0307 P0006
SFTON P0307
MOVL C00399 BC00399 V=66.7 PL=0
SFTOF
'------------------------
'W56A P
'------------------------
SFTOF
MOVJ C00400 BC00400 VJ=30.00
MOVL C00401 BC00401 V=133.3 PL=0
REFP 3 C00402 BC00402
CALL JOB:SEARCH-R1
SET P0308 P0006
SFTON P0308
MOVL C00403 BC00403 V=66.7 PL=0
REFP 3 C00404 BC00404
CALL JOB:SEARCH-R1
SET P0308 P0006
SFTON P0308
MOVL C00405 BC00405 V=66.7 PL=0
SFTOF
'------------------------
SFTOF
MOVJ C00406 BC00406 VJ=30.00
MOVL C00407 BC00407 V=250.0
MOVL C00408 BC00408 V=66.7 PL=0
REFP 3 C00409 BC00409
CALL JOB:SEARCH-R1
SET P0309 P0006
SFTON P0309
MOVL C00410 BC00410 V=66.7 PL=0
REFP 3 C00411 BC00411
CALL JOB:SEARCH-R1
SET P0309 P0006
SFTON P0309
MOVL C00412 BC00412 V=66.7 PL=0
SFTOF
'------------------------
SFTOF
MOVJ C00413 BC00413 VJ=5.00
MOVJ C00414 BC00414 VJ=20.00
MOVL C00415 BC00415 V=116.7 PL=0
REFP 3 C00416 BC00416
CALL JOB:SEARCH-R1
SET P0310 P0006
SFTON P0310
MOVL C00417 BC00417 V=66.7 PL=0
REFP 3 C00418 BC00418
CALL JOB:SEARCH-R1
SET P0310 P0006
SFTON P0310
MOVL C00419 BC00419 V=66.7 PL=0
SFTOF
'------------------------
'W55A L
'------------------------
SFTOF
MOVL C00420 BC00420 V=250.0
MOVJ C00421 BC00421 VJ=10.00
MOVL C00422 BC00422 V=66.7 PL=0
REFP 3 C00423 BC00423
CALL JOB:SEARCH-R1
SET P0311 P0006
SFTON P0311
MOVL C00424 BC00424 V=66.7 PL=0
REFP 3 C00425 BC00425
CALL JOB:SEARCH-R1
SET P0311 P0006
SFTON P0311
MOVL C00426 BC00426 V=66.7 PL=0
SFTOF
SFTOF
'------------------------
'W55A P
'------------------------
SFTOF
MOVL C00427 BC00427 V=250.0
MOVL C00428 BC00428 V=166.7
MOVL C00429 BC00429 V=66.7 PL=0
REFP 3 C00430 BC00430
CALL JOB:SEARCH-R1
SET P0312 P0006
SFTON P0312
MOVL C00431 BC00431 V=66.7 PL=0
REFP 3 C00432 BC00432
CALL JOB:SEARCH-R1
SET P0312 P0006
SFTON P0312
MOVL C00433 BC00433 V=66.7 PL=0
MOVL C00434 BC00434 V=166.7
SFTOF
MOVL C00435 BC00435 V=250.0
MOVJ C00436 BC00436 VJ=20.00
MOVJ C00437 BC00437 VJ=30.00
MOVJ C00438 BC00438 VJ=20.00
MOVJ C00439 BC00439 VJ=20.00
MOVJ C00440 BC00440 VJ=20.00
MOVJ C00441 BC00441 VJ=20.00
MOVJ C00442 BC00442 VJ=20.00
'------------------------
'LEWA STRONA PROFIL GORA
'------------------------
MOVJ C00443 BC00443 VJ=10.00
'------------------------
SFTOF
MOVJ C00444 BC00444 VJ=10.00
MOVL C00445 BC00445 V=66.7 PL=0
REFP 3 C00446 BC00446
CALL JOB:SEARCH-R1
SET P0349 P0006
SFTON P0349
MOVL C00447 BC00447 V=66.7 PL=0
REFP 3 C00448 BC00448
CALL JOB:SEARCH-R1
SET P0349 P0006
SFTON P0349
MOVL C00449 BC00449 V=66.7 PL=0
SFTOF
MOVJ C00450 BC00450 VJ=10.00
MOVJ C00451 BC00451 VJ=10.00
'------------------------
'W55B P
'------------------------
SFTOF
MOVL C00452 BC00452 V=66.7 PL=0
REFP 3 C00453 BC00453
CALL JOB:SEARCH-R1
SET P0350 P0006
SFTON P0350
MOVL C00454 BC00454 V=66.7 PL=0
REFP 3 C00455 BC00455
CALL JOB:SEARCH-R1
SET P0350 P0006
SFTON P0350
MOVL C00456 BC00456 V=66.7 PL=0
SFTOF
'------------------------
'W52B L
'------------------------
SFTOF
MOVJ C00457 BC00457 VJ=20.00
MOVJ C00458 BC00458 VJ=20.00
MOVL C00459 BC00459 V=150.0
MOVL C00460 BC00460 V=66.7 PL=0
REFP 3 C00461 BC00461
CALL JOB:SEARCH-R1
SET P0351 P0006
SFTON P0351
MOVL C00462 BC00462 V=66.7 PL=0
REFP 3 C00463 BC00463
CALL JOB:SEARCH-R1
SET P0351 P0006
SFTON P0351
MOVL C00464 BC00464 V=66.7 PL=0
SFTOF
'------------------------
'W52B P
'------------------------
SFTOF
MOVJ C00465 BC00465 VJ=30.00
MOVL C00466 BC00466 V=116.7 PL=0
REFP 3 C00467 BC00467
CALL JOB:SEARCH-R1
SET P0352 P0006
SFTON P0352
MOVL C00468 BC00468 V=66.7 PL=0
REFP 3 C00469 BC00469
CALL JOB:SEARCH-R1
SET P0352 P0006
SFTON P0352
MOVL C00470 BC00470 V=66.7 PL=0
SFTOF
'------------------------
'W56B L
'------------------------
SFTOF
MOVJ C00471 BC00471 VJ=30.00
MOVL C00472 BC00472 V=116.7 PL=0
REFP 3 C00473 BC00473
CALL JOB:SEARCH-R1
SET P0353 P0006
SFTON P0353
MOVL C00474 BC00474 V=66.7 PL=0
REFP 3 C00475 BC00475
CALL JOB:SEARCH-R1
SET P0353 P0006
SFTON P0353
MOVL C00476 BC00476 V=66.7 PL=0
SFTOF
'------------------------
'W56B P
'------------------------
SFTOF
MOVJ C00477 BC00477 VJ=30.00
MOVL C00478 BC00478 V=116.7 PL=0
REFP 3 C00479 BC00479
CALL JOB:SEARCH-R1
SET P0354 P0006
SFTON P0354
MOVL C00480 BC00480 V=66.7 PL=0
REFP 3 C00481 BC00481
CALL JOB:SEARCH-R1
SET P0354 P0006
SFTON P0354
MOVL C00482 BC00482 V=66.7 PL=0
SFTOF
'------------------------
'W53B L
'------------------------
SFTOF
MOVJ C00483 BC00483 VJ=30.00
MOVL C00484 BC00484 V=116.7 PL=0
REFP 3 C00485 BC00485
CALL JOB:SEARCH-R1
SET P0355 P0006
SFTON P0355
MOVL C00486 BC00486 V=66.7 PL=0
REFP 3 C00487 BC00487
CALL JOB:SEARCH-R1
SET P0355 P0006
SFTON P0355
MOVL C00488 BC00488 V=66.7 PL=0
SFTOF
'------------------------
'W53B P
'------------------------
SFTOF
MOVJ C00489 BC00489 VJ=30.00
MOVL C00490 BC00490 V=116.7 PL=0
REFP 3 C00491 BC00491
CALL JOB:SEARCH-R1
SET P0356 P0006
SFTON P0356
MOVL C00492 BC00492 V=66.7 PL=0
REFP 3 C00493 BC00493
CALL JOB:SEARCH-R1
SET P0356 P0006
SFTON P0356
MOVL C00494 BC00494 V=66.7 PL=0
SFTOF
'------------------------
'W50B L
'------------------------
SFTOF
MOVJ C00495 BC00495 VJ=30.00
MOVL C00496 BC00496 V=116.7 PL=0
REFP 3 C00497 BC00497
CALL JOB:SEARCH-R1
SET P0357 P0006
SFTON P0357
MOVL C00498 BC00498 V=66.7 PL=0
REFP 3 C00499 BC00499
CALL JOB:SEARCH-R1
SET P0357 P0006
SFTON P0357
MOVL C00500 BC00500 V=66.7 PL=0
SFTOF
'------------------------
'W50B P
'------------------------
SFTOF
MOVJ C00501 BC00501 VJ=30.00
MOVL C00502 BC00502 V=116.7 PL=0
REFP 3 C00503 BC00503
CALL JOB:SEARCH-R1
SET P0358 P0006
SFTON P0358
MOVL C00504 BC00504 V=66.7 PL=0
REFP 3 C00505 BC00505
CALL JOB:SEARCH-R1
SET P0358 P0006
SFTON P0358
MOVL C00506 BC00506 V=66.7 PL=0
SFTOF
'------------------------
'W54B L
'------------------------
SFTOF
MOVJ C00507 BC00507 VJ=30.00
MOVL C00508 BC00508 V=116.7 PL=0
REFP 3 C00509 BC00509
CALL JOB:SEARCH-R1
SET P0359 P0006
SFTON P0359
MOVL C00510 BC00510 V=66.7 PL=0
REFP 3 C00511 BC00511
CALL JOB:SEARCH-R1
SET P0359 P0006
SFTON P0359
MOVL C00512 BC00512 V=66.7 PL=0
SFTOF
'------------------------
'W54B P
'------------------------
SFTOF
MOVJ C00513 BC00513 VJ=30.00
MOVL C00514 BC00514 V=116.7 PL=0
REFP 3 C00515 BC00515
CALL JOB:SEARCH-R1
SET P0360 P0006
SFTON P0360
MOVL C00516 BC00516 V=66.7 PL=0
REFP 3 C00517 BC00517
CALL JOB:SEARCH-R1
SET P0360 P0006
SFTON P0360
MOVL C00518 BC00518 V=166.7 PL=0
SFTOF
'------------------------
'W51B L
'------------------------
'------------------------
SFTOF
MOVL C00519 BC00519 V=150.0
MOVL C00520 BC00520 V=66.7 PL=0
REFP 3 C00521 BC00521
CALL JOB:SEARCH-R1
SET P0361 P0006
SFTON P0361
MOVL C00522 BC00522 V=66.7 PL=0
REFP 3 C00523 BC00523
CALL JOB:SEARCH-R1
SET P0361 P0006
SFTON P0361
MOVL C00524 BC00524 V=83.3
MOVL C00525 BC00525 V=133.3 PL=0
REFP 3 C00526 BC00526
CALL JOB:SEARCH-R1
SET P0361 P0006
SFTON P0361
SFTOF
MOVL C00527 BC00527 V=83.3
MOVJ C00528 BC00528 VJ=20.00
MOVJ C00529 BC00529 VJ=30.00
MOVJ C00530 BC00530 VJ=10.00
MOVJ C00531 BC00531 VJ=40.00
'**********************
'**********************
'POCZATEK SPAWANIA BOKI
'**********************
'**********************
MOVJ C00532 BC00532 VJ=30.00
MOVJ C00533 BC00533 VJ=20.00
'**********************
'W50A
'**********************
MOVL C00534 BC00534 V=250.0
SFTON P0304
MOVL C00535 BC00535 V=83.3 PL=0
SFTOF
MACRO1 MJ#(0) ARGF10
ARCON
SFTON P0303
MOVL C00536 BC00536 V=10.8
ARCOF
SFTOF
MOVL C00537 BC00537 V=250.0
'W13B
MOVJ C00538 BC00538 VJ=20.00
MOVJ C00539 BC00539 VJ=40.00
MOVJ C00540 BC00540 VJ=20.00
MOVJ C00541 BC00541 VJ=20.00
MOVJ C00542 BC00542 VJ=20.00
'**********************
'W50B
'**********************
MOVL C00543 BC00543 V=250.0
SFTON P0357
MOVL C00544 BC00544 V=166.7 PL=0
SFTOF
MACRO1 MJ#(0) ARGF10
ARCON
SFTON P0358
MOVL C00545 BC00545 V=10.8
ARCOF
SFTOF
MOVL C00546 BC00546 V=250.0
MOVJ C00547 BC00547 VJ=20.00
MOVJ C00548 BC00548 VJ=20.00
MOVJ C00549 BC00549 VJ=20.00
MOVJ C00550 BC00550 VJ=20.00
'**********************
'W51A
'**********************
MOVL C00551 BC00551 V=416.7
SFTON P0299
MOVL C00552 BC00552 V=166.7 PL=0
SFTOF
MACRO1 MJ#(0) ARGF10
ARCON
SFTON P0299
COMM MOVL C00553 BC00553 V=10.8
MOVL C00554 BC00554 V=10.8
ARCOF
MOVL C00555 BC00555 V=166.7
MOVL C00556 BC00556 V=133.3 PL=0
ARCON
MOVL C00557 BC00557 V=8.3
ARCOF
SFTOF
MOVL C00558 BC00558 V=200.0
MOVJ C00559 BC00559 VJ=30.00
MOVJ C00560 BC00560 VJ=30.00
MOVJ C00561 BC00561 VJ=30.00
MOVJ C00562 BC00562 VJ=30.00
MOVJ C00563 BC00563 VJ=30.00
'**********************
'W51B
'**********************
MOVL C00564 BC00564 V=416.7
MOVL C00565 BC00565 V=416.7
SFTON P0361
MOVL C00566 BC00566 V=166.7 PL=0
SFTOF
MACRO1 MJ#(0) ARGF10
ARCON
SFTON P0361
MOVL C00567 BC00567 V=10.8
MOVL C00568 BC00568 V=10.8
ARCOF
MOVL C00569 BC00569 V=166.7
MACRO1 MJ#(0) ARGF9
MOVL C00570 BC00570 V=166.7 PL=0
ARCON
MOVL C00571 BC00571 V=8.3
ARCOF
SFTOF
MOVL C00572 BC00572 V=166.7
MOVL C00573 BC00573 V=250.0
MOVJ C00574 BC00574 VJ=30.00
MOVJ C00575 BC00575 VJ=30.00
MOVJ C00576 BC00576 VJ=30.00
MOVJ C00577 BC00577 VJ=40.00
MOVJ C00578 BC00578 VJ=40.00
MOVJ C00579 BC00579 VJ=20.00
MOVJ C00580 BC00580 VJ=20.00
MOVJ C00581 BC00581 VJ=20.00
MOVJ C00582 BC00582 VJ=20.00
MOVJ C00583 BC00583 VJ=20.00
'**********************
'W52A
'**********************
SFTON P0310
MOVL C00584 BC00584 V=250.0
MOVL C00585 BC00585 V=83.3 PL=0
SFTOF
MACRO1 MJ#(0) ARGF10
ARCON
SFTON P0309
MOVL C00586 BC00586 V=10.8
ARCOF
SFTOF
MOVL C00587 BC00587 V=333.3
MOVJ C00588 BC00588 VJ=30.00
MOVJ C00589 BC00589 VJ=30.00
MOVJ C00590 BC00590 VJ=30.00
MOVJ C00591 BC00591 VJ=30.00
MOVJ C00592 BC00592 VJ=30.00
MOVJ C00593 BC00593 VJ=20.00
MOVJ C00594 BC00594 VJ=20.00
MOVJ C00595 BC00595 VJ=20.00
'**********************
'52B
'**********************
MOVL C00596 BC00596 V=250.0
SFTON P0351
MOVL C00597 BC00597 V=83.3 PL=0
SFTOF
MACRO1 MJ#(0) ARGF10
ARCON
SFTON P0352
MOVL C00598 BC00598 V=10.8
ARCOF
MOVL C00599 BC00599 V=333.3
SFTOF
MOVJ C00600 BC00600 VJ=20.00
MOVJ C00601 BC00601 VJ=30.00
MOVJ C00602 BC00602 VJ=30.00
'**********************
'W53A
'**********************
MOVJ C00603 BC00603 VJ=30.00
MOVJ C00604 BC00604 VJ=30.00
MOVJ C00605 BC00605 VJ=10.00
'**********************
'W53A
'**********************
SFTON P0306
MOVL C00606 BC00606 V=250.0
MOVL C00607 BC00607 V=83.3 PL=0
SFTOF
MACRO1 MJ#(0) ARGF10
ARCON
SFTON P0305
MOVL C00608 BC00608 V=10.8
ARCOF
SFTOF
MOVL C00609 BC00609 V=250.0
MOVJ C00610 BC00610 VJ=30.00
MOVJ C00611 BC00611 VJ=30.00
MOVJ C00612 BC00612 VJ=30.00
MOVJ C00613 BC00613 VJ=30.00
MOVJ C00614 BC00614 VJ=30.00
MOVJ C00615 BC00615 VJ=30.00
MOVL C00616 BC00616 V=250.0
'**********************
'W53B
'**********************
SFTON P0355
MOVL C00617 BC00617 V=250.0
MOVL C00618 BC00618 V=83.3 PL=0
SFTOF
MACRO1 MJ#(0) ARGF10
ARCON
SFTON P0356
MOVL C00619 BC00619 V=10.8
ARCOF
SFTOF
MOVL C00620 BC00620 V=333.3
MOVJ C00621 BC00621 VJ=30.00
MOVJ C00622 BC00622 VJ=30.00
MOVJ C00623 BC00623 VJ=30.00
MOVJ C00624 BC00624 VJ=30.00
'**********************
'W54A
'**********************
SFTON P0302
MOVL C00625 BC00625 V=250.0
MOVL C00626 BC00626 V=83.3 PL=0
SFTOF
MACRO1 MJ#(0) ARGF10
ARCON
SFTON P0301
MOVL C00627 BC00627 V=10.8
ARCOF
SFTOF
MOVL C00628 BC00628 V=333.3
MOVJ C00629 BC00629 VJ=20.00
MOVJ C00630 BC00630 VJ=30.00
MOVJ C00631 BC00631 VJ=30.00
MOVJ C00632 BC00632 VJ=30.00
MOVJ C00633 BC00633 VJ=30.00
'**********************
'W54B
'**********************
SFTON P0359
MOVL C00634 BC00634 V=250.0
MOVL C00635 BC00635 V=83.3 PL=0
SFTOF
MACRO1 MJ#(0) ARGF10
ARCON
SFTON P0360
MOVL C00636 BC00636 V=10.8
ARCOF
MOVL C00637 BC00637 V=333.3
SFTOF
MOVJ C00638 BC00638 VJ=30.00
MOVJ C00639 BC00639 VJ=30.00
MOVJ C00640 BC00640 VJ=30.00
MOVJ C00641 BC00641 VJ=40.00
MOVJ C00642 BC00642 VJ=40.00
MOVJ C00643 BC00643 VJ=10.00
MOVJ C00644 BC00644 VJ=10.00
MOVJ C00645 BC00645 VJ=10.00
MOVJ C00646 BC00646 VJ=15.00
MOVJ C00647 BC00647 VJ=15.00
MOVJ C00648 BC00648 VJ=15.00
MOVJ C00649 BC00649 VJ=15.00
'**********************
'W55A
'**********************
SFTON P0311
MOVL C00650 BC00650 V=166.7 PL=0
SFTOF
MACRO1 MJ#(0) ARGF10
ARCON
SFTON P0312
MOVL C00651 BC00651 V=10.8
MOVL C00652 BC00652 V=10.8
ARCOF
SFTOF
MOVL C00653 BC00653 V=150.0
MOVJ C00654 BC00654 VJ=10.00
MOVJ C00655 BC00655 VJ=10.00
MOVJ C00656 BC00656 VJ=10.00
MOVJ C00657 BC00657 VJ=10.00
MOVJ C00658 BC00658 VJ=10.00
MOVJ C00659 BC00659 VJ=10.00
MOVJ C00660 BC00660 VJ=30.00
MOVJ C00661 BC00661 VJ=30.00
MOVJ C00662 BC00662 VJ=20.00
MOVJ C00663 BC00663 VJ=30.00
MOVJ C00664 BC00664 VJ=20.00
MOVJ C00665 BC00665 VJ=20.00
MOVJ C00666 BC00666 VJ=30.00
MOVJ C00667 BC00667 VJ=20.00
MOVJ C00668 BC00668 VJ=20.00
'**********************
'W55B
'**********************
SFTON P0350
MOVL C00669 BC00669 V=333.3
MOVL C00670 BC00670 V=166.7 PL=0
SFTOF
MACRO1 MJ#(0) ARGF10
ARCON
SFTON P0349
MOVL C00671 BC00671 V=10.8
MOVL C00672 BC00672 V=10.8
ARCOF
SFTOF
MOVL C00673 BC00673 V=66.7
MOVJ C00674 BC00674 VJ=10.00
MOVJ C00675 BC00675 VJ=20.00
MOVJ C00676 BC00676 VJ=20.00
MOVJ C00677 BC00677 VJ=20.00
MOVJ C00678 BC00678 VJ=30.00
MOVJ C00679 BC00679 VJ=50.00
MOVJ C00680 BC00680 VJ=50.00
MOVJ C00681 BC00681 VJ=40.00
MOVJ C00682 BC00682 VJ=20.00
'**********************
'W56A
'**********************
SFTON P0308
MOVL C00683 BC00683 V=333.3
MOVL C00684 BC00684 V=166.7 PL=0
SFTOF
MACRO1 MJ#(0) ARGF10
ARCON
SFTON P0307
MOVL C00685 BC00685 V=10.8
ARCOF
SFTOF
MOVL C00686 BC00686 V=333.3
MOVJ C00687 BC00687 VJ=20.00
MOVJ C00688 BC00688 VJ=30.00
MOVJ C00689 BC00689 VJ=30.00
MOVJ C00690 BC00690 VJ=30.00
'**********************
'W56B
'**********************
SFTON P0353
MOVL C00691 BC00691 V=250.0
MOVL C00692 BC00692 V=166.7 PL=0
SFTOF
MACRO1 MJ#(0) ARGF10
ARCON
SFTON P0354
MOVL C00693 BC00693 V=10.8
ARCOF
SFTOF
MOVL C00694 BC00694 V=333.3
MOVJ C00695 BC00695 VJ=30.00
MOVJ C00696 BC00696 VJ=30.00
MOVJ C00697 BC00697 VJ=30.00
CALL JOB:MOVE_OUT_OF_TUNNEL
CALL JOB:R1-HOME
END
